        |   ph7 = p[p0x-d1, p0y, p0z-0.05, 0, 0, 0]
        | 
        |   # add the vertical touch points
        |   if pointtop[2] == 0:
        |     ph2up = p[ph2[0], ph2[1], ph2[2]+d3, ph2[3], ph2[4], ph2[5]]
        |     ph4up = p[ph4[0], ph4[1], ph4[2]+d3, ph4[3], ph4[4], ph4[5]]
        |   elif pointtop[2] > p0z + 0.914: # 0.914m = 36 inches
        |     ph2up = p[ph2[0], ph2[1], p0z + 0.914, ph2[3], ph2[4], ph2[5]]
        |     ph4up = p[ph4[0], ph4[1], p0z + 0.914, ph4[3], ph4[4], ph4[5]]
        |   else:
        |     ph2up = p[ph2[0], ph2[1], pointtop[2], ph2[3], ph2[4], ph2[5]]
        |     ph4up = p[ph4[0], ph4[1], pointtop[2], ph4[3], ph4[4], ph4[5]]
        |   end
        |   ret = struct(ph1=ph1, ph2=ph2, ph3=ph3, ph4=ph4, ph5=ph5, ph6=ph6, ph7=ph7, ph2up=ph2up, ph4up=ph4up)
        |   is_robot_at_reachable_spot(point0, ret)
        |   return ret
        | end
        | 
        | # this function checks whether the touchpoints are reachable AKA is the robot positioned in the right spot
        | # if everything looks good, it continues.
        | # if it detects a problem, it infinite loops a popup
        | def is_robot_at_reachable_spot(point0, struct_touchpoints):
        |   # first, check whether the corner is too low to the ground that the bottom homing will hit the ground (z < -400)
        |   lc_height = get_lift_column_height_condensed()
        |   # total height = zeroed lift column height (41.25 inches) (1.04775 m) plus lift column height plus robot relative height
        |   totalheight = 1.04775 + lc_height + point0[2]
        |   if totalheight < 1.04775 - 0.400:
        |     # bad
        |     popuptext = "Tank Corner is too low to the ground. Collisions will occur. Stop Program and raise tank. "
        |     # infinite loop
        |     while 1==1:
        |       popup(popuptext, title="Robot Positioning Warning",blocking=True)
        |     end
        |   end
        | 
        | 
        | 
        |   # next, check whether the touchpoints are reachable
        |   allvalid = check_structofpoints_validity(struct_touchpoints)
        |   if not allvalid:
        | 
        |     # then unreachable
        |     # generate message
        |     listproblems = ""
        |     listnames = ["ph1", "ph2", "ph3", "ph4", "ph5", "ph6", "ph7", "ph2up", "ph4up"]
        |     i = 0
        |     structlength = 9
        |     while i < structlength:
        |       curr = struct_touchpoints[i]
        |       valid = get_inverse_kin_has_solution(curr)
        |       if not valid:
        |         listproblems = listproblems + listnames[i]
        |       end
        |       i = i + 1
        |     end
        |     # display
        |     popuptext = "Robot is too far from tank corner. Cannot reach some necessary positions. Stop Program and move robot closer. " + listproblems
        |     # infinite loop
        |     while 1==1:
        |       popup(popuptext, title="Robot Positioning Warning",blocking=True)
        |     end
        |   end
        | 
        | end
        | 
        | # this function takes a struct of points as an argument, and checks whether every point in the list is reachable using get_inverse_kin_has_solution()
        | # this function does NOT check for weird twists or joint limits
        | # inputstruct must contain only points
        | # it returns true if all points are valid. it returns false if any points are valid
        | # a list of length 0 indicates that all points are valid
        | def check_structofpoints_validity(inputstruct):
        |   # next, check whether the touchpoints are reachable
        |   structlength = length(inputstruct)
        |   i = 0
        |   allvalid = True
        |   while i < structlength:
        |     curr = inputstruct[i]
        |     valid = get_inverse_kin_has_solution(curr)
        |     if not valid:
        |       return False
        |     end
        |     i = i + 1
        |   end
        |   return True
        | end
        | 
        | # checks the validity of all points during a left weld
        | # takes 2 arguments: struct1 (struct1[0] has to contain pointintersect) and struct2 (contains all the points (9) of the weld path)
        | def check_validity_left(struct1, struct2):
        |   #first, check whether robot is too close
        |   pointintersect = struct1[0]
        |   # next, check if the corner is too close to the robot to do a left around weld (complex but approximately X > -1300)
        |   # if y < 0, then x < -1300. if y < 480, then y > (1300+x)*8. if y > 480, then y > (1235+x)*4 + 500
        |   toocloseleftweld = False
        |   if pointintersect[1] < 0:
        |     if pointintersect[0] > -1.300:
        |       toocloseleftweld = True
        |     end
        |   elif pointintersect[1] < 0.480:
        |     if pointintersect[1] < (1.300 + pointintersect[0])*8:
        |       toocloseleftweld = True
        |     end
        |   else:
        |     if pointintersect[1] < (1.235 + pointintersect[0])*4 + 0.500:
        |       toocloseleftweld = True
        |     end
        |   end
        |   if toocloseleftweld:
        |     # bad
        |     popuptext = "Robot is too close to tank corner. Collisions may occur. Stop Program and move robot farther. "
        |     # infinite loop
        |     while 1==1:
        |       popup(popuptext, title="Robot Positioning Warning",blocking=True)
        |     end
        |   end
        | 
        |   #next, check whether all the points in the weldpath are valid
        |   structlength = 9
        |   i = 0
        |   allvalid = True
        |   listproblems = ""
        |   listnames = ["point1", "point2", "point4", "point5", "point_1", "point_2", "point_3", "point_4", "point_5"]
        |   while i < structlength:
        |     curr = struct2[i]
        |     valid = get_inverse_kin_has_solution(curr)
        |     if not valid:
        |       allvalid = False
        |       listproblems = listproblems + listnames[i]
        |     end
        |     i = i + 1
        |   end
        | 
        |   if not allvalid:
        |     # display
        |     popuptext = "Robot is too far from tank corner. Cannot reach some necessary positions. Stop Program and move robot closer. " + listproblems
        |     # infinite loop
        |     while 1==1:
        |       popup(popuptext, title="Robot Positioning Warning",blocking=True)
        |     end
        |   end
        | 
        |   # check whether the path involves weird turns or joint limits. currently just checks the first position
        |   p_prev = [-0.021118, -1.26292, 2.43578, 5.07088, -2.29912, 1.53362] #last point of left weld prerotate
        |   joints_1 = get_inverse_kin(struct2[0], p_prev) # struct2[0] is point1
        |   allGood = True
        |   i = 0
        |   structlength = 6
        |   while i < structlength:
        |     joint_curr = joints_1[i]
        |     # check for anything that exceeds joint limits
        |     degreesmax = 360 * pi / 180
        |     if joint_curr > degreesmax or joint_curr < degreesmax * -1:
        |       allGood = False
        |     end
        |     # check for anything that is significantly different than the aligned approach. could indicate a twist is needed. we dont want that
        |     maxdifference = 150 * pi / 180
        |     difference = joint_curr - p_prev[i]
        |     if difference > maxdifference or difference * -1 > maxdifference:
        |       allGood = False
        |     end
        |     i = i + 1
        |   end
        | 
        |   if not allGood:
        |     # call lift column extend function
        |     struct2 = floor_corner_lift_column_extend_left(struct2)
        | 
        |   end
        | 
        |   # return struct2 back
        |   return struct2
        | end
        | 
        | # checks the validity of all points during a right weld
        | def check_validity_right(struct1, struct2):
        |   # first, check whether the right pivot will bonk itself
        |   pointintersect = struct1[0]
        |   heading1 = struct1[1] # this is the direction that the welder will face when doing the right side of the box
        | 
        |   #first, check whether the heading is just too far offset
        |   # more than 15 degrees off of 45 is too much
        |   # normal heading is 216 degrees
        |   #201 degrees to 231 degrees
        |   heading1degrees = heading1 * 180 / pi
        |   if heading1degrees < 201 or heading1degrees > 231 :
        |     # then out of range
        |     popuptext = "Robot is not aligned at a 45 degree angle of corner (15 degree leeway). Collisions may occur. Stop Program and align robot. heading1degrees=" + str_cat("",heading1degrees)
        |     # infinite loop
        |     while 1==1:
        |       popup(popuptext, title="Robot Positioning Warning",blocking=True)
        |     end
        |   end
        | 
        |   #TODO: add the checks for whether x is too close, given the heading
        |   # add checks for whether x is too close, given the heading
        |   # different equations for whether heading offset > 5 degrees or less (inc. negative)
        |   headingoffset = heading1degrees - 216
        |   if headingoffset < 5:
        |     # then calculate a and b
        |     a = 0.4584 + -0.02369 * headingoffset
        |     b = (-1151.4 + 13.83 * headingoffset) / 1000
        |     # check whether x > a*y+b
        |     if pointintersect[0] > a * pointintersect[1] + b:
        |       # bad
        |       popuptext = "Robot is too close to tank corner or not at the right angle. Collisions may occur. Stop Program and align robot. "
        |       # infinite loop
        |       while 1==1:
        |         popup(popuptext, title="Robot Positioning Warning",blocking=True)
        |       end
        |     end
        |   else:
        |     # headingoffset > 5 degrees
        |     if pointintersect[1] < 0:
        |       if pointintersect[0] > -1150.0 / 1000.0:
        |         #bad
        |         popuptext = "Robot is too close to tank corner. Collisions may occur. Stop Program and align robot. "
        |         # infinite loop
        |         while 1==1:
        |           popup(popuptext, title="Robot Positioning Warning",blocking=True)
        |         end
        |       end
        |     else:
        |       # if x > .7736 y - 1101.9 then bad
        |       if pointintersect[0] > 0.7736 * pointintersect[1] - 1101.9 / 1000:
        |         popuptext = "Robot is too close to tank corner. Collisions may occur. Stop Program and align robot. "
        |         # infinite loop
        |         while 1==1:
        |           popup(popuptext, title="Robot Positioning Warning",blocking=True)
        |         end
        |       end
        |     end
        |   end
        | 
        |   #next, check whether all the points in the weldpath are valid
        |   structlength = 9
        |   i = 0
        |   allvalid = True
        |   listproblems = ""
        |   listnames = ["point1", "point2", "point4", "point5", "point_1", "point_2", "point_3", "point_4", "point_5"]
        |   while i < structlength:
        |     curr = struct2[i]
        |     valid = get_inverse_kin_has_solution(curr)
        |     if not valid:
        |       allvalid = False
        |       listproblems = listproblems + listnames[i]
        |     end
        |     i = i + 1
        |   end
        | 
        |   if not allvalid:
        |     # display
        |     popuptext = "Robot is too far from tank corner. Cannot reach some necessary positions. Stop Program and move robot closer. " + listproblems
        |     # infinite loop
        |     while 1==1:
        |       popup(popuptext, title="Robot Positioning Warning",blocking=True)
        |     end
        |   end
        | 
        |   # check whether the path involves weird turns or joint limits. currently just checks the first position
        |   p_prev = [-1.13307, -1.48911, 2.84785, 4.92357, -4.89059, 1.57184] #last point of right weld prerotate
        |   joints_1 = get_inverse_kin(struct2[0], p_prev) # struct2[0] is point1
        |   allGood = True
        |   i = 0
        |   structlength = 6
        |   while i < structlength:
        |     joint_curr = joints_1[i]
        |     # check for anything that exceeds joint limits
        |     degreesmax = 360 * pi / 180
        |     if joint_curr > degreesmax or joint_curr < degreesmax * -1:
        |       allGood = False
        |     end
        |     # check for anything that is significantly different than the aligned approach. could indicate a twist is needed. we dont want that
        |     maxdifference = 150 * pi / 180
        |     difference = joint_curr - p_prev[i]
        |     if difference > maxdifference or difference * -1 > maxdifference:
        |       allGood = False
        |     end
        |     i = i + 1
        |   end
        | 
        |   if not allGood:
        |     struct2 = floor_corner_lift_column_extend_right(struct2)
        |   end
        | 
        |   # return struct2 back
        |   return struct2
        | end
        | 
        | def floor_corner_lift_column_extend_right(struct2):
        |   # we know that p1 cannot be accessed without a twist
        |   # calculate the height needed to get to p1
        |   liftcolumnincrement = 2.0 # mm
        |   enoughHeightAdded = False
        |   liftColumnHeightTest = 0
        |   while not enoughHeightAdded:
        |     liftColumnHeightTest = liftColumnHeightTest + liftcolumnincrement
        |     # set the orig_joints for p1. p1 demo was joint angles of [-0.45, -31.79, 56.47, 333.06, -130.98, 87.87] (degrees)
        |     # which equals [-0.007853981633974475, -0.5548401692089968, 0.985587428601197, 5.812993606692308, -2.28603225426217, 1.5336208137274159]
        |     orig_joints = [-0.007853981633974475, -0.5548401692089968, 0.985587428601197, 5.812993606692308, -2.28603225426217, 1.5336208137274159]
        |     # get the modified point:
        |     origp1 = struct2[0]
        |     testp1 = p[origp1[0], origp1[1], origp1[2] - liftColumnHeightTest / 1000.0, origp1[3], origp1[4], origp1[5]]
        |     testpa1 = p[origp1[0]+0.05, origp1[1]+0.05, origp1[2] - liftColumnHeightTest / 1000, origp1[3], origp1[4], origp1[5]]
        |     enoughHeightAdded = can_pose_be_reached_without_twist(testp1, orig_joints) and can_pose_be_reached_without_twist(testpa1, orig_joints)
        |   end
        | 
        |   origp2 = struct2[1]
        |   testp2 = p[origp2[0], origp2[1], origp2[2] - liftColumnHeightTest / 1000.0, origp2[3], origp2[4], origp2[5]]
        |   origp4 = struct2[2]
        |   testp4 = p[origp4[0], origp4[1], origp4[2] - liftColumnHeightTest / 1000, origp4[3], origp4[4], origp4[5]]
        |   origp5 = struct2[3]
        |   testp5 = p[origp5[0], origp5[1], origp5[2] - liftColumnHeightTest / 1000, origp5[3], origp5[4], origp5[5]]
        | 
        | 
        | 
        |   liftcolumnzneeded = liftColumnHeightTest
        |   ret = struct(point1=testp1,point2=testp2,point4=testp4,point5=testp5,point_1=struct2[4],point_2=struct2[5],point_3=struct2[6],point_4=struct2[7],point_5=struct2[8])
        |   return ret
        | 
        | end
        | 
        | # this function gets called if you are doing a left floor corner extended, and the top is too high to reach (twists, etc.)
        | # this function takes the struct2 of weld points and modifies them (by subtracting from z) until the first weld point is reachable.
        | # it determines the height that the lift column needs to raise to make the first point reachable
        | # it then checks whether that height will allow the other points to be reachable
        | # if its all good, it sets the global variable liftcolumnzneeded, modifies struct2's points, and returns struct2
        | # if its not all good, then it displays an error message popup.
        | def floor_corner_lift_column_extend_left(struct2):
        |   # we know that p1 cannot be accessed without a twist
        |   # calculate the height needed to get to p1
        |   liftcolumnincrement = 2 # mm
        |   enoughHeightAdded = False
        |   liftColumnHeightTest = 0
        |   while not enoughHeightAdded:
        |     liftColumnHeightTest = liftColumnHeightTest + liftcolumnincrement
        |     # set the orig_joints for p1. p1 demo was joint angles of [-0.45, -31.79, 56.47, 333.06, -130.98, 87.87] (degrees)
        |     # which equals [-0.007853981633974475, -0.5548401692089968, 0.985587428601197, 5.812993606692308, -2.28603225426217, 1.5336208137274159]
        |     orig_joints = [-0.007853981633974475, -0.5548401692089968, 0.985587428601197, 5.812993606692308, -2.28603225426217, 1.5336208137274159]
        |     # get the modified point:
        |     origp1 = struct2[0]
        |     testp1 = p[origp1[0], origp1[1], origp1[2] - liftColumnHeightTest / 1000, origp1[3], origp1[4], origp1[5]]
        |     enoughHeightAdded = can_pose_be_reached_without_twist(testp1, orig_joints)
        |   end
        | 
        |   # check whether the other 3 points are valid
        |   valid = True
        |   # get the modified point
        |   origp2 = struct2[1]
        |   testp2 = p[origp2[0], origp2[1], origp2[2] - liftColumnHeightTest / 1000, origp2[3], origp2[4], origp2[5]]
        |   # p2 demo was joint angles of [-0.45, -21.2, 56.98, 321.95, -130.97, 87.85] (degrees)
        |   # which equals [-0.007853981633974475, -0.3700098014227975, 0.9944886077863679, 5.619087526795738, -2.285857721336971, 1.5332717478770168]
        |   orig_joints = [-0.007853981633974475, -0.3700098014227975, 0.9944886077863679, 5.619087526795738, -2.285857721336971, 1.5332717478770168]
        |   valid = valid and can_pose_be_reached_without_twist(testp2, orig_joints)
        |   # get the modified point
        |   origp4 = struct2[2]
        |   testp4 = p[origp4[0], origp4[1], origp4[2] - liftColumnHeightTest / 1000, origp4[3], origp4[4], origp4[5]]
        |   # p4 demo was joint angles of [-8.62, -43.23, 99.53, 213.86, -89.19, 40.78] (degrees)
        |   # which equals [-0.15044738152191103, -0.7545058356371478, 1.7371262045099545, 3.7325611383150696, -1.556659159853741, 0.7117452689632868]
        |   orig_joints = [-0.15044738152191103, -0.7545058356371478, 1.7371262045099545, 3.7325611383150696, -1.556659159853741, 0.7117452689632868]
        |   valid = valid and can_pose_be_reached_without_twist(testp4, orig_joints)
        |   # get the modified point
        |   origp5 = struct2[3]
        |   testp5 = p[origp5[0], origp5[1], origp5[2] - liftColumnHeightTest / 1000, origp5[3], origp5[4], origp5[5]]
        |   # p5 demo was joint angles of [-0.59, -34.36, 77.71, 226.7, -89.18, 48.81] (degrees)
        |   # which equals [-0.010297442586766533, -0.5996951309852511, 1.356295361724792, 3.9566614142711405, -1.5564846269285415, 0.8518952078984314]
        |   orig_joints = [-0.010297442586766533, -0.5996951309852511, 1.356295361724792, 3.9566614142711405, -1.5564846269285415, 0.8518952078984314]
        |   valid = valid and can_pose_be_reached_without_twist(testp5, orig_joints)
        | 
        |   if not valid:
        |     # display
        |     popuptext = "Top of Weld is too high above robot. Cannot reach some necessary positions. Stop Program and try again with a lower top point. "
        |     # infinite loop
        |     while 1==1:
        |       popup(popuptext, title="Robot Positioning Warning",blocking=True)
        |     end
        |   else:
        |     liftcolumnzneeded = liftColumnHeightTest
        |     ret = struct(point1=testp1,point2=testp2,point4=testp4,point5=testp5,point_1=struct2[4],point_2=struct2[5],point_3=struct2[6],point_4=struct2[7],point_5=struct2[8])
        |     return ret
        |   end
        | end
        | 
        | # this function calculates whether a given pose can be reached, and if it can, whether it requires a wrist twist (from the seed joint angles)
        | # arguments are target pose (p[x,y,z,rx,ry,rz]) and orig_joints which is the 6 joint angles of a pose that is close by the target pose and has the desired joint angles
        | # returns true if the pose is valid and requires no twist. If pose is valid but requires a twist, returns false. If pose is invalid, returns false.
        | def can_pose_be_reached_without_twist(pose, orig_joints):
        |   # first, determine if the pose is valid
        |   valid = get_inverse_kin_has_solution(pose)
        |   if not valid:
        |     return False
        |   end
        |   joints_1 = get_inverse_kin(pose, orig_joints)
        |   #iterate through the 6 joints
        |   allGood = True
        |   i = 0
        |   structlength = 6
        |   while i < structlength:
        |     joint_curr = joints_1[i]
        |     # check for anything that exceeds joint limits
        |     degreesmax = 360 * pi / 180
        |     if joint_curr > degreesmax or joint_curr < degreesmax * -1:
        |       allGood = False
        |     end
        |     # check for anything that is significantly different than the aligned approach. could indicate a twist is needed. we dont want that
        |     maxdifference = 150 * pi / 180
        |     difference = joint_curr - orig_joints[i]
        |     if difference > maxdifference or difference * -1 > maxdifference:
        |       allGood = False
        |     end
        |     i = i + 1
        |   end
        |   return allGood
        | end
        | 
        | # this function sends a signal to turn extrusion on
        | def turn_extrusion_on():
        |   # flush the channel
        |   resp0 = send_serial_signal(["u", "r", "?"])
        |   # send the signal
        |   resp1 = send_serial_signal(["u", "R", "1"])
        |   # if resp <> "uR1"
        |   if resp1 != [252,82,49]:
        |     # turn off extrusion and heating. inform calvin
        |     resp2 = send_serial_signal(["u", "R", "0"])
        |     resp3 = send_serial_signal(["u", "H", "0"])
        |     popuptext = "Error code encountered while trying to start extrusion. Find Calvin. "
        |     while 1==1:
        |       popup(popuptext, title="Extrusion Error Code",blocking=True)
        |       popup(resp1, blocking=True)
        |     end
        |   end
        | end
        | 
        | # this function sends a signal and receives a response
        | # signal is a list of 3 strings, 1 character each. first is u. second is the next character. third is final character
        | def send_serial_signal(signal):
        |   signal2char = signal[1]
        |   signal3char = signal[2]
        |   listsignal = [252, get_corr_number(signal2char), get_corr_number(signal3char)]
        |   resp1 = WTSerialBridge.send_command("/dev/ttyUSB0",1200, 8, "None", "One", "None", 1000, "None", "None", listsignal, True)
        |   return resp1
        | end
        | 
        | # this function converts a letter into its ascii number
        | def get_corr_number(letter):
        |   if letter == "A":
        |     return 65
        |   elif letter == "H":
        |     return 72
        |   elif letter == "R":
        |     return 82
        |   elif letter == "M":
        |     return 77
        |   elif letter == "E":
        |     return 69
        |   elif letter == "a":
        |     return 97
        |   elif letter == "b":
        |     return 98
        |   elif letter == "h":
        |     return 104
        |   elif letter == "r":
        |     return 114
        |   elif letter == "s":
        |     return 115
        |   elif letter == "m":
        |     return 109
        |   elif letter == "0":
        |     return 48
        |   elif letter == "1":
        |     return 49
        |   elif letter == "2":
        |     return 50
        |   elif letter == "3":
        |     return 51
        |   elif letter == "4":
        |     return 52
        |   elif letter == "5":
        |     return 53
        |   elif letter == "6":
        |     return 54
        |   elif letter == "7":
        |     return 55
        |   elif letter == "8":
        |     return 56
        |   elif letter == "9":
        |     return 57
        |   elif letter == "?":
        |     return 63
        |   end
        | end
        | 
        | # this function checks whether the welder is in the ready state.
        | # to be called at the beginning of Main Program
        | def welder_state_ready():
        |   # flush the channel
        |   resp0 = send_serial_signal(["u", "s", "?"])
        |   # send the signal
        |   resp1 = send_serial_signal(["u", "s", "?"])
        |   # if resp1 == [252,115,49] (us1) then it is ready. otherwise, it is not
        |   if resp1 != [252,115,49]:
        |     popuptext = "Welder is not ready for extrusion. Follow the instructions to start heating welder. "
        |     while 1==1:
        |       popup(popuptext, title="Welder Not Ready",blocking=True)
        |     end
        |   end
        | 
        | end
        | 
        | def get_lift_column_height():
        |   # begin: URCap Program Node
        |   #   Source: MachineLogic for Universal Robots, 3.1.7, Vention Inc.
        |   #   Type: MachineLogic for Universal Robots
        |   #$ 5 "MachineLogic Get Position"
        |   while isVentionMovementBusyMachineMotion1==True:
        |     sleep(0.05)
        |   end
        |   if(isVentionMovementBusyMachineMotion1 == False):
        |     isVentionMovementBusyMachineMotion1 = True
        |     socket_send_string("estop/status;", "MachineMotion1")
        |     temp_estop_var_vention = socket_read_string("MachineMotion1",timeout=15)
        |     while(temp_estop_var_vention=="estop/status true"):
        |       if temp_estop_var_vention=="estop/status true":
        |         sendStringWithTimeout("estop/systemreset/request","Ack estop/systemreset/request;","MachineMotion1")
        |       end
        |       socket_send_string("estop/status;", "MachineMotion1")
        |       temp_estop_var_vention = socket_read_string("MachineMotion1",timeout=15)
        |       if temp_estop_var_vention=="estop/status true":
        |         popup("MachineMotion in estop, make sure you have all emergency modules released manually. If you continue the system will try to reset MachineMotion automatically.",blocking=True)
        |       end
        |     end
        |   else:
        |     popup("resource is being used already: MachineMotion1")
        |     halt
        |   end
        |   socket_send_string("GET im_get_controller_pos_axis_1;", "MachineMotion1")
        |   temp_drive = socket_read_ascii_float(1, "MachineMotion1",timeout=15)
        |   global var_1 = temp_drive[1]
        |   isVentionMovementBusyMachineMotion1 = False
        |   sleep(0.03)
        |   # end: URCap Program Node
        | end
        | 
        | def get_lift_column_height_condensed():
        |   socket_send_string("GET im_get_controller_pos_axis_1;", "MachineMotion1")
        |   temp_drive = socket_read_ascii_float(1, "MachineMotion1",timeout=15)
        |   ret = temp_drive[1]
        |   return ret
        | end
  'list possible points'
  Folder robot 1 moves
    If 1≟2
      MoveJ speed 60 deg/s, acceleration 80 deg/s^2 (useActiveTCP=true optimoveEnabled=false optiMoveSpeed=0.3 optiMoveAcceleration=0.09) feature=Base
        Waypoint r1_ek_oldhome: TCP in base x=397.38 y=356.254 z=319.821 mm, rx=2.3163 ry=2.0576 rz=0.0741 rad; joints [-198.126, -117.851, 133.303, -13.009, -11.422, -6.035] deg; TCP offset x=-5.49 y=-328 z=106.39 mm, rx=1.2092 ry=-1.2092 rz=1.2092 rad
        Waypoint r1_ek_extrude: TCP in base x=454.852 y=405.449 z=64.015 mm, rx=2.3168 ry=2.0514 rz=0.0767 rad; joints [-187.624, -89.406, 141.395, -19.732, -0.818, -36.116] deg
        Waypoint r1_ek_front: TCP in base x=439.065 y=405.452 z=65.996 mm, rx=2.3168 ry=2.0514 rz=0.0766 rad; joints [-187.962, -93.321, 143.386, -27.168, -1.131, -26.752] deg
        Waypoint r1_ek_middle: TCP in base x=419.01 y=404.851 z=65.995 mm, rx=2.3096 ry=2.0447 rz=0.0891 rad; joints [-188.553, -97.485, 146.002, -33.769, -1.69, -19.324] deg
        Waypoint r1_ek_middle2: TCP in base x=417.012 y=405.435 z=65.003 mm, rx=2.3169 ry=2.0513 rz=0.0766 rad; joints [-188.493, -97.025, 145.794, -33.21, -1.638, -19.415] deg
        Waypoint r1_ek_bottom: TCP in base x=413.072 y=405.431 z=68 mm, rx=2.3168 ry=2.0513 rz=0.0767 rad; joints [-188.596, -97.887, 146.02, -33.517, -1.738, -18.475] deg
        Waypoint r1_ek_end: TCP in base x=389.999 y=405.444 z=68.005 mm, rx=2.3169 ry=2.0514 rz=0.0766 rad; joints [-189.248, -101.07, 148.002, -36.337, -2.38, -14.447] deg
  Folder robot 2 moves
    If 1≟2
      MoveJ speed 60 deg/s, acceleration 80 deg/s^2 (useActiveTCP=true optimoveEnabled=false optiMoveSpeed=0.3 optiMoveAcceleration=0.09) feature=Base
        Waypoint r2_ek_oldhome: TCP in base x=397.38 y=356.254 z=319.821 mm, rx=2.3163 ry=2.0576 rz=0.0741 rad; joints [-198.308, -118.162, 133.451, -12.562, -11.515, -6.325] deg; TCP offset x=-9.5 y=-328 z=105.73 mm, rx=1.2092 ry=-1.2092 rz=1.2092 rad
        SuppressedNode
          Waypoint Waypoint_1: TCP in base x=612.886 y=429.305 z=100.477 mm, rx=1.8619 ry=2.4807 rz=0.0957 rad; joints [-182.793, -81.736, 125.569, -42.478, -18.966, -5.44] deg
        Waypoint r2_ek_extrude: TCP in base x=612.886 y=429.305 z=100.477 mm, rx=2.15 ry=2.2258 rz=0.0874 rad; joints [-183.316, -85.158, 129.692, -39.696, -5.262, -8.969] deg
        Waypoint r2_ek_front: TCP in base x=556.405 y=429.305 z=76.984 mm, rx=-2.1704 ry=-2.2682 rz=-0.0159 rad; joints [-183.513, -85.623, 132.794, -41.666, -5.994, -5.809] deg
        Waypoint r2_ek_middle: TCP in base x=550.034 y=429.305 z=76.254 mm, rx=-2.1704 ry=-2.2682 rz=-0.0159 rad; joints [-183.554, -85.983, 133.283, -41.831, -6.035, -5.773] deg
        Waypoint r2_ek_bottom: TCP in base x=546.595 y=429.305 z=80.868 mm, rx=-2.1704 ry=-2.2682 rz=-0.0159 rad; joints [-183.576, -86.513, 133.34, -41.373, -6.058, -5.758] deg
        Waypoint r2_ek_end: TCP in base x=537.335 y=429.305 z=80.868 mm, rx=-2.1704 ry=-2.2682 rz=-0.0159 rad; joints [-183.639, -87.118, 134.001, -41.482, -6.12, -5.705] deg
  'detemine correct points for which robot'
  If robot_number≟1
    Folder robot1 positions
      ek_oldhome := r1_ek_oldhome_p
      ek_extrude := r1_ek_extrude_p
      ek_front := r1_ek_front_p
      ek_middle := r1_ek_middle_p
      ek_middle2 := r1_ek_middle2_p
      ek_bottom := r1_ek_bottom_p
      ek_end := r1_ek_end_q
  ElseIf robot_number≟2
    Folder robot1 positions
      ek_oldhome := r2_ek_oldhome_p
      ek_extrude := r2_ek_extrude_p
      ek_front := r2_ek_front_p
      ek_middle := r2_ek_middle_p
      ek_middle2 := r2_ek_middle_p
      ek_bottom := r2_ek_bottom_p
      ek_end := r2_ek_end_q
  'start of program'
  SuppressedNode
    SafeHome (positionOptionType=SPEED_AND_ACCELERATION speed=1.047198 acceleration=1.396263 nextMotionTime=2)
  Set NoAction tcp=pretend_welder
  MoveJ speed 60 deg/s, acceleration 80 deg/s^2 (useActiveTCP=true optimoveEnabled=false optiMoveSpeed=0.3 optiMoveAcceleration=0.09) feature=Base
    SuppressedNode
      Waypoint r1_ek_oldhome: TCP in base x=397.38 y=356.254 z=319.821 mm, rx=2.3163 ry=2.0576 rz=0.0741 rad; joints [-198.126, -117.851, 133.303, -13.009, -11.422, -6.035] deg; TCP offset x=-5.49 y=-328 z=106.39 mm, rx=1.2092 ry=-1.2092 rz=1.2092 rad
    Waypoint Variable (Variable): variable=ek_oldhome
    'above waypoint is home'
  'move above bucket'
  MoveJ speed 60 deg/s, acceleration 80 deg/s^2 (useActiveTCP=true optimoveEnabled=false optiMoveSpeed=0.3 optiMoveAcceleration=0.09) feature=Base
    SuppressedNode
      Waypoint r1_ek_extrude: TCP in base x=454.852 y=405.449 z=64.015 mm, rx=2.3168 ry=2.0514 rz=0.0767 rad; joints [-187.624, -89.406, 141.395, -19.732, -0.818, -36.116] deg
    Waypoint Variable (Variable): variable=ek_extrude
  'extrude out a foot'
  SuppressedNode
    Script: turn_extrusion_on()
  URCap WireTank Serial (WireTank Serial, WireTank, LLC) dataModel(NODE_TITLE=Serial Bridge uR1, Command=[252,82,49], QUERY=false, byte_array=true, OUTPUT_ENTRY=Static, Variable(key=OUTPUT_VARIABLE, variable(name=HwResp)))
  Set DigitalOutput pin=digital_out[0]; digitalValue=1
  Wait Sleep waitTime=24
  URCap WireTank Serial (WireTank Serial, WireTank, LLC) dataModel(QUERY=false, NODE_TITLE=Serial Bridge uR0, Command=[252,82,48], byte_array=true, OUTPUT_ENTRY=Static, Variable(key=OUTPUT_VARIABLE, variable(name=HwResp)))
  Wait Sleep waitTime=1
  Set DigitalOutput pin=digital_out[0]; digitalValue=0
  'slice'
  MoveL speed 30 mm/s, acceleration 50 mm/s^2 (useActiveTCP=true optimoveEnabled=false optiMoveSpeed=0.3 optiMoveAcceleration=0.09) feature=Base
    SuppressedNode
      Waypoint r1_ek_front: TCP in base x=439.065 y=405.452 z=65.996 mm, rx=2.3168 ry=2.0514 rz=0.0766 rad; joints [-187.962, -93.321, 143.386, -27.168, -1.131, -26.752] deg
    SuppressedNode
      Waypoint r1_ek_middle: TCP in base x=419.01 y=404.851 z=65.995 mm, rx=2.3096 ry=2.0447 rz=0.0891 rad; joints [-188.553, -97.485, 146.002, -33.769, -1.69, -19.324] deg
    SuppressedNode
      Waypoint r1_ek_middle2: TCP in base x=417.012 y=405.435 z=65.003 mm, rx=2.3169 ry=2.0513 rz=0.0766 rad; joints [-188.493, -97.025, 145.794, -33.21, -1.638, -19.415] deg
    SuppressedNode
      Waypoint r1_ek_bottom: TCP in base x=413.072 y=405.431 z=68 mm, rx=2.3168 ry=2.0513 rz=0.0767 rad; joints [-188.596, -97.887, 146.02, -33.517, -1.738, -18.475] deg
    SuppressedNode
      Waypoint r1_ek_end: TCP in base x=389.999 y=405.444 z=68.005 mm, rx=2.3169 ry=2.0514 rz=0.0766 rad; joints [-189.248, -101.07, 148.002, -36.337, -2.38, -14.447] deg
    Waypoint Variable (Variable): variable=ek_front
    Waypoint Variable (Variable): variable=ek_middle
    Waypoint Variable (Variable): variable=ek_middle2
    Waypoint Variable (Variable): variable=ek_bottom
    Waypoint Variable (Variable): variable=ek_end
  MoveJ speed 60 deg/s, acceleration 80 deg/s^2 (useActiveTCP=true optimoveEnabled=false optiMoveSpeed=0.3 optiMoveAcceleration=0.09) feature=Base
    SuppressedNode
      Waypoint r1_ek_oldhome: TCP in base x=397.38 y=356.254 z=319.821 mm, rx=2.3163 ry=2.0576 rz=0.0741 rad; joints [-198.126, -117.851, 133.303, -13.009, -11.422, -6.035] deg
    Waypoint Variable (Variable): variable=ek_oldhome
    'above waypoint is home'
  SuppressedNode
    SafeHome (positionOptionType=SPEED_AND_ACCELERATION speed=1.047198 acceleration=1.396263 nextMotionTime=2)
SubProgram align_tcp_forward (keepSynchronizedWithDisk=false) programFile=/programs/align_tcp_forward.urp
  'this program aligns the tcp parallel to the y direction'
  cp := get_actual_tcp_pose()
  aligned_y_pose := p[cp[0],cp[1],cp[2],0,-1.570796,0]
  MoveJ speed 60 deg/s, acceleration 80 deg/s^2 (useActiveTCP=true optimoveEnabled=false optiMoveSpeed=0.3 optiMoveAcceleration=0.09) feature=Base
    Waypoint Variable (Variable): variable=aligned_y_pose
SubProgram align_tcp_up (keepSynchronizedWithDisk=false) programFile=/programs/align_tcp_up.urp
  'this program aligns the tcp parallel to the y direction'
  cp := get_actual_tcp_pose()
  aligned_y_pose := p[cp[0],cp[1],cp[2],0,0,0]
  MoveJ speed 60 deg/s, acceleration 80 deg/s^2 (useActiveTCP=true optimoveEnabled=false optiMoveSpeed=0.3 optiMoveAcceleration=0.09) feature=Base
    Waypoint Variable (Variable): variable=aligned_y_pose
SubProgram align_for_step (keepSynchronizedWithDisk=false) programFile=/programs/align_for_step.urp
  'first move block is unnecessay and bad'
  SuppressedNode
    MoveJ speed 60 deg/s, acceleration 80 deg/s^2 (useActiveTCP=true optimoveEnabled=false optiMoveSpeed=0.3 optiMoveAcceleration=0.09) feature=Base
      'belowis oldhome'
      Waypoint Waypoint_1: TCP in base x=397.354 y=356.263 z=319.809 mm, rx=2.3163 ry=2.0576 rz=0.0741 rad; joints [-198.308, -118.162, 133.452, -12.561, -11.517, -6.326] deg; TCP offset x=-9.5 y=-328 z=105.73 mm, rx=1.2092 ry=-1.2092 rz=1.2092 rad
      SuppressedNode
        Waypoint Waypoint_2: TCP in base x=102.072 y=804.129 z=-21.158 mm, rx=-1.0098 ry=-2.9661 rz=0.0347 rad; joints [-131.791, -72.228, 126.432, -52.794, -4.122, -0.058] deg
      SuppressedNode
        Waypoint Waypoint_3: TCP in base x=-481.576 y=738.776 z=-387.745 mm, rx=-0.0268 ry=3.1371 rz=-0.1325 rad; joints [-88.373, -42.244, 121.849, -79.055, 0.705, 4.289] deg
      Waypoint Waypoint_4: TCP in base x=-790.625 y=220.046 z=-730.503 mm, rx=-0.9425 ry=2.9648 rz=-0.1356 rad; joints [-49.775, -15.59, 117.776, -102.401, 4.996, 5.448] deg
      Waypoint Waypoint_5: TCP in base x=-802.158 y=237.168 z=-730.663 mm, rx=0.8868 ry=-2.4516 rz=0.2829 rad; joints [-61.24, 14.733, 101.407, -222.645, 33.575, 110.967] deg
      Waypoint Waypoint_6: TCP in base x=-687.678 y=589.975 z=-233.622 mm, rx=-0.3444 ry=-1.0001 rz=-2.0808 rad; joints [-61.24, 14.733, 101.407, -222.645, 33.575, -30.853] deg
      SuppressedNode
        Waypoint goalpt: TCP in base x=-796.965 y=229.005 z=-75.004 mm, rx=0 ry=0 rz=-2.526 rad; joints [-49.775, -15.59, 117.776, -102.401, 4.996, -179.788] deg
      Waypoint goalpt2: TCP in base x=-1080.054 y=352.633 z=-86.722 mm, rx=0.0341 ry=-0.0008 rz=-2.631 rad; joints [-41.761, 5.394, 77.547, 101.81, -19.08, -4.137] deg
      Waypoint dummythere: TCP in base x=-1288.589 y=229.005 z=-75.004 mm, rx=0 ry=0 rz=-2.526 rad; joints [-29.748, -12.575, 79.071, -66.58, 25.031, -179.927] deg
  'second one is good'
  SuppressedNode
    MoveJ speed 60 deg/s, acceleration 80 deg/s^2 (useActiveTCP=true optimoveEnabled=false optiMoveSpeed=0.3 optiMoveAcceleration=0.09) feature=Base
      Waypoint goalpt2: TCP in base x=-1080.054 y=352.633 z=-86.722 mm, rx=0.0341 ry=-0.0008 rz=-2.631 rad; joints [-41.761, 5.394, 77.547, 101.81, -19.08, -4.137] deg
  'above was for wrong weldpath'
  SuppressedNode
    Folder savepoints
      MoveJ speed 60 deg/s, acceleration 80 deg/s^2 (useActiveTCP=true optimoveEnabled=false optiMoveSpeed=0.3 optiMoveAcceleration=0.09) feature=Base
        Waypoint leftstart: TCP in base x=-1168.534 y=251.879 z=303.712 mm, rx=-1.4388 ry=-0.6695 rz=0.6003 rad; joints [-161.388, -128.913, -89.606, -145.038, 61.894, 92.57] deg
  SuppressedNode
    MoveJ speed 60 deg/s, acceleration 80 deg/s^2 (useActiveTCP=true optimoveEnabled=false optiMoveSpeed=0.3 optiMoveAcceleration=0.09) feature=Base
      'final point before pa1'
      Waypoint Waypoint_7: TCP in base x=-913.411 y=251.879 z=303.712 mm, rx=-1.2351 ry=-1.1043 rz=1.0523 rad; joints [-156.391, -105.358, -132.178, -128.187, 33.298, 95.672] deg
      'oldhome'
      Waypoint Waypoint_8: TCP in base x=397.354 y=356.263 z=319.809 mm, rx=2.3163 ry=2.0576 rz=0.0741 rad; joints [-198.308, -118.162, 133.452, -12.561, -11.517, -6.326] deg
  MoveJ speed 60 deg/s, acceleration 80 deg/s^2 (useActiveTCP=true optimoveEnabled=false optiMoveSpeed=0.3 optiMoveAcceleration=0.09) feature=Base
    'from oldhome, actual path'
    SuppressedNode
      Waypoint Waypoint_9: TCP in base x=683.137 y=304.628 z=775.294 mm, rx=1.9572 ry=1.7212 rz=0.4516 rad; joints [-193.46, -116.682, 102.732, -25.933, -6.334, 5.47] deg
    SuppressedNode
      Waypoint Waypoint_10: TCP in base x=-197.847 y=491.143 z=1723.576 mm, rx=-0.0125 ry=0.2444 rz=1.7982 rad; joints [-175.692, -50.406, -94.795, -74.947, 12.663, 48.707] deg
    Waypoint Waypoint_1: TCP in base x=-557.589 y=419.56 z=1207.727 mm, rx=-0.5026 ry=-0.0558 rz=1.8139 rad; joints [-165.719, -50.766, -121.227, -102.266, 18.039, 76.633] deg
    SuppressedNode
      Waypoint Waypoint_12: TCP in base x=-793.876 y=251.879 z=303.712 mm, rx=-1.2351 ry=-1.1043 rz=1.0523 rad; joints [-150.736, -98.884, -141.754, -124.357, 38.932, 94.772] deg
  MoveJ speed 60 deg/s, acceleration 80 deg/s^2 (useActiveTCP=true optimoveEnabled=false optiMoveSpeed=0.3 optiMoveAcceleration=0.09) feature=Base
    SuppressedNode
      Waypoint Waypoint_12: TCP in base x=-793.876 y=251.879 z=303.712 mm, rx=-1.2351 ry=-1.1043 rz=1.0523 rad; joints [-150.736, -98.884, -141.754, -124.357, 38.932, 94.772] deg
    Waypoint Waypoint_3: TCP in base x=-479.957 y=297.468 z=291.375 mm, rx=-0.7812 ry=-1.774 rz=1.7129 rad; joints [-222.662, -82.07, -155.488, -122.893, -85.563, 87.81] deg
  SuppressedNode
    Folder dummy points
      'for seeing if it goes to each side correctly'
      MoveJ speed 60 deg/s, acceleration 80 deg/s^2 (useActiveTCP=true optimoveEnabled=false optiMoveSpeed=0.3 optiMoveAcceleration=0.09) feature=Base
        'right side weld'
        Waypoint Waypoint_15: TCP in base x=-1072.479 y=376.012 z=295.965 mm, rx=-0.7812 ry=-1.774 rz=1.7129 rad; joints [-196.962, -109.785, -121.389, -129.338, -59.875, 88.022] deg
      MoveL speed 10 mm/s, acceleration 50 mm/s^2 (useActiveTCP=true optimoveEnabled=false optiMoveSpeed=0.3 optiMoveAcceleration=0.09) feature=Base
        Waypoint Waypoint_14: TCP in base x=-1156.816 y=297.468 z=291.375 mm, rx=-0.7812 ry=-1.774 rz=1.7129 rad; joints [-189.786, -111.954, -118.346, -130.254, -52.7, 88.101] deg
SubProgram retreat_from_step (keepSynchronizedWithDisk=false) programFile=/programs/retreat_from_step.urp
  SuppressedNode
    Folder dummy points
      MoveJ speed 60 deg/s, acceleration 80 deg/s^2 (useActiveTCP=true optimoveEnabled=false optiMoveSpeed=0.3 optiMoveAcceleration=0.09) feature=Base
        'right side end points'
        Waypoint Waypoint_1: TCP in base x=-1253.519 y=364.13 z=-67.585 mm, rx=0.018 ry=0.0176 rz=0.7803 rad; joints [-179.095, -181.39, -36.733, -141.231, 46.177, 180.871] deg
        Waypoint Waypoint_3: TCP in base x=-1253.519 y=364.13 z=-129.324 mm, rx=0.018 ry=0.0176 rz=0.7803 rad; joints [-179.093, -185.871, -31.706, -141.776, 46.177, 180.869] deg
      MoveJ speed 60 deg/s, acceleration 80 deg/s^2 (useActiveTCP=true optimoveEnabled=false optiMoveSpeed=0.3 optiMoveAcceleration=0.09) feature=Base
        'left side end points'
        Waypoint Waypoint_4: TCP in base x=-1258.059 y=209.945 z=-65.388 mm, rx=0.0265 ry=-0.0276 rz=2.2505 rad; joints [-170.66, -165.644, -86.102, -104.787, -29.65, 176.354] deg
        Waypoint Waypoint_5: TCP in base x=-1258.059 y=209.945 z=-131.718 mm, rx=0.0265 ry=-0.0276 rz=2.2505 rad; joints [-170.658, -169.867, -82.992, -103.675, -29.649, 176.354] deg
  MoveJ speed 60 deg/s, acceleration 80 deg/s^2 (useActiveTCP=true optimoveEnabled=false optiMoveSpeed=0.3 optiMoveAcceleration=0.09) feature=Base
    Waypoint Waypoint_16: TCP in base x=-670.966 y=326.422 z=-178.215 mm, rx=0.0098 ry=0.0257 rz=1.6447 rad; joints [-167.814, -172.971, -116.48, -67.413, 7.981, 178.204] deg
  MoveJ speed 60 deg/s, acceleration 80 deg/s^2 (useActiveTCP=true optimoveEnabled=false optiMoveSpeed=0.3 optiMoveAcceleration=0.09) feature=Base
    Waypoint Waypoint_17: TCP in base x=-635.85 y=491.712 z=259.684 mm, rx=-0.4995 ry=-0.7883 rz=1.854 rad; joints [-203.235, -128.315, -150.467, -80.055, -46.632, 133.613] deg
    Waypoint Waypoint_18: TCP in base x=-479.957 y=297.468 z=291.375 mm, rx=-0.7812 ry=-1.774 rz=1.7129 rad; joints [-222.662, -82.07, -155.488, -122.893, -85.563, 87.81] deg
  MoveJ speed 60 deg/s, acceleration 80 deg/s^2 (useActiveTCP=true optimoveEnabled=false optiMoveSpeed=0.3 optiMoveAcceleration=0.09) feature=Base
    Waypoint Waypoint_20: TCP in base x=-557.589 y=419.56 z=1207.727 mm, rx=-0.5026 ry=-0.0558 rz=1.8139 rad; joints [-165.719, -50.766, -121.227, -102.266, 18.039, 76.633] deg
  SafeHome (positionOptionType=SPEED_AND_ACCELERATION speed=1.047198 acceleration=1.396263 nextMotionTime=2)
SubProgram Corner_Homing_45 (keepSynchronizedWithDisk=false) programFile=/programs/Corner Homing 45.urp
  'Use this program when tool is already positioned close to corner at 45deg'
  'tool flange will seek all 3 sides. will save those 5 locs in p__'
  Set NoAction tcp=pretend_w_top
  'dummy move below for debug'
  SuppressedNode
    SafeHome (positionOptionType=SPEED_AND_ACCELERATION speed=1.047198 acceleration=1.396263 nextMotionTime=2)
  SuppressedNode
    MoveJ speed 60 deg/s, acceleration 80 deg/s^2 (useActiveTCP=true optimoveEnabled=false optiMoveSpeed=0.3 optiMoveAcceleration=0.09) feature=Base
      Waypoint Waypoint_1: TCP in base x=-726.76 y=313.857 z=-3.219 mm, rx=-0.1302 ry=-1.6605 rz=-0.1403 rad; joints [-65.067, -50.619, 153.092, -93.35, 35.027, 81.724] deg; TCP offset x=0 y=0 z=246 mm, rx=0 ry=0 rz=0 rad
      Waypoint Waypoint_2: TCP in base x=-1013.668 y=283.774 z=13.404 mm, rx=-0.1302 ry=-1.6605 rz=-0.1403 rad; joints [-36.803, -53.188, 133.142, -74.065, 63.057, 86.565] deg
  Wait Sleep waitTime=1
  tp := get_actual_tcp_pose()
  SuppressedNode
    Script file /programs/analyze_touchpoints.script
      | # this file creates the function for analyzing touchpoints
      | # define pi
      | pi = 3.1415926535
      | 
      | # this is the main entry point for calculations.
      | # it takes in the 5 points, analyzes the shape of the box, and then calculates path points and returns them
      | # specifically for Down, Over, then Around (DOtA)
      | # specifically for right-sided boxes (vertical weld on right side of edge)
      | def main_calculate_right(p11, p12, p21, p22, p3, p13, p23, chamferover):
      |     struct1 = analyze_touchpoints_only(p11, p12, p21, p22, p3)
      |     list1 = analyze_vertical_touchpoints(p11, p12, p13, p21, p22, p23, p3)
      |     struct2 = calculate_DOtA_points_right(struct1, list1, chamferover)
      |     validity = check_validity_right(struct1, struct2)
      |     return struct2
      | end
      | 
      | # this is the main entry point for calculations.
      | # it takes in the 5 points, analyzes the shape of the box, and then calculates path points and returns them
      | # specifically for Down, Over, then Around (DOtA)
      | # specifically for left-sided boxes (vertical weld on left side of edge)
      | def main_calculate_left(p11, p12, p21, p22, p3, p13, p23, chamferover):
      |     struct1 = analyze_touchpoints_only(p11, p12, p21, p22, p3)
      |     list1 = analyze_vertical_touchpoints(p11, p12, p13, p21, p22, p23, p3)
      |     struct2 = calculate_DOtA_points_left(struct1, list1, chamferover)
      |     validity = check_validity_left(struct1, struct2)
      |     return struct2
      | end
      | 
      | # this is the main entry point for calculations, for Floor Corner Extended.
      | # it takes in the 7 touchpoints, analyzes the shape of the box.
      | # takes in the user defined point for the top of the weld (tcp_pose_top) and then calculates path points
      | # loopingly tries to calculate the extension along the sidewall that fulfills get_inverse_kin_has_solution() and provides the farthest extension possible
      | # returns the pathpoints
      | # specifically for Down, Over, then Around (DOtA)
      | # specifically for right-sided boxes (vertical weld on right side of edge)
      | def main_calculate_right_extended(p11, p12, p21, p22, p3, p13, p23, chamferover, tcp_pose_top):
      |     struct1 = analyze_touchpoints_only(p11, p12, p21, p22, p3)
      |     list1 = analyze_vertical_touchpoints(p11, p12, p13, p21, p22, p23, p3)
      |     struct2 = calculate_DOtA_points_right_extended(struct1, list1, chamferover, tcp_pose_top)
      |     validity = check_validity_right(struct1, struct2)
      |     return struct2
      | end
      | 
      | # this is the main entry point for calculations, for Floor Corner Extended.
      | # it takes in the 7 touchpoints, analyzes the shape of the box.
      | # takes in the user defined point for the top of the weld (tcp_pose_top) and then calculates path points
      | # loopingly tries to calculate the extension along the sidewall that fulfills get_inverse_kin_has_solution() and provides the farthest extension possible
      | # returns the pathpoints
      | # specifically for Down, Over, then Around (DOtA)
      | # specifically for left-sided boxes (vertical weld on left side of edge)
      | def main_calculate_left_extended(p11, p12, p21, p22, p3, p13, p23, chamferover, tcp_pose_top):
      |     struct1 = analyze_touchpoints_only(p11, p12, p21, p22, p3)
      |     list1 = analyze_vertical_touchpoints(p11, p12, p13, p21, p22, p23, p3)
      |     struct2 = calculate_DOtA_points_left_extended(struct1, list1, chamferover, tcp_pose_top)
      |     validity = check_validity_left(struct1, struct2)
      |     return struct2
      | end
      | 
      | # it takes 5 arguments as points
      | # it returns a struct containing: (pointintersect, pointapproach1, pointapproach2, point1, point2, point3, point4, point5, pointreturn1, heading1, heading2, heading3, path2r1, path2r2, path2l1, path2l2)
      | # specifically for Around then Up (AtU)
      | def analyze_touchpoints(p11, p12, p21, p22, p3):
      |   # FIND THE INTERSECTION
      |   # comment get the z
      |   zcoord=p3[2]
      | 
      |   # get the raw points from the first line
      |   l1p1x=p11[0]
      |   l1p1y=p11[1]
      |   l1p2x=p12[0]
      |   l1p2y=p12[1]
      | 
      |   # equate the first line in 2d space
      |   ml1 = (l1p2y-l1p1y) / (l1p2x-l1p1x)
      | 
      |   # b = y - mx
      |   bl1 = l1p1y - ml1 * l1p1x
      | 
      |   # get the raw points from the second line
      |   l2p1x=p21[0]
      |   l2p1y=p21[1]
      |   l2p2x=p22[0]
      |   l2p2y=p22[1]
      | 
      |   # equate the second line in 2d space
      |   ml2 = (l2p2y-l2p1y) / (l2p2x-l2p1x)
      | 
      |   # b = y - mx
      |   bl2 = l2p1y - ml2 * l2p1x
      | 
      | 
      |   # find the intersection of the two lines
      |   # m1x+b1 = m2x+b2
      |   # m1x - m2x = b2 - b1
      |   # x = (b2-b1) / (m1-m2)
      |   xintersect = (bl2-bl1) / (ml1-ml2)
      |   yintersect = ml1 * xintersect + bl1
      | 
      |   #FIND THE VECTORS
      |   #define a vector from the intersection to the second point on the first line
      |   l1delxfull = l1p2x - xintersect
      |   l1delyfull = l1p2y - yintersect
      | 
      |   l1delmag = sqrt(l1delxfull*l1delxfull + l1delyfull*l1delyfull)
      | 
      |   l1delxunit = l1delxfull / l1delmag
      |   l1delyunit = l1delyfull / l1delmag
      | 
      |   #define a vector from the intersection to the second point on the second line
      |   l2delxfull = l2p2x - xintersect
      |   l2delyfull = l2p2y - yintersect
      | 
      |   l2delmag = sqrt(l2delxfull*l2delxfull + l2delyfull*l2delyfull)
      | 
      |   l2delxunit = l2delxfull / l2delmag
      |   l2delyunit = l2delyfull / l2delmag
      | 
      |   # FIND THE FOUR POINTS ON THE LINES
      |   # find locations 8 inches away from  intersect point
      |   # CONST
      |   welddistance = 8
      |   roundoverdistance = 0.05
      |   zup = .375
      |   # inches
      |   wd = welddistance * 25.4 / 1000
      |   rod = roundoverdistance * 25.4 / 1000
      |   zup = zup * 25.4 / 1000
      | 
      |   # now we have the unit vector. extend the weld distance from the intersection
      |   x = xintersect + l1delxunit * wd
      |   y = yintersect + l1delyunit * wd
      |   z = zcoord + zup
      | 
      |   point1 = p[x,y,z,1.570796,0,0] # dummy orientation for now
      | 
      |   x = xintersect + l1delxunit * rod
      |   y = yintersect + l1delyunit * rod
      | 
      |   point2 = p[x,y,z,1.570796,0,0]
      | 
      |   # now we have the unit vector. extend the weld distance from the intersection
      |   x = xintersect + l2delxunit * wd
      |   y = yintersect + l2delyunit * wd
      | 
      |   point5 = p[x,y,z,0,-1.570796,0]
      | 
      |   x = xintersect + l2delxunit * rod
      |   y = yintersect + l2delyunit * rod
      | 
      |   point4 = p[x,y,z,0,-1.570796,0]
      | 
      |   #DEFINE APPROACH POINTS
      |   pointintersect = p[xintersect,yintersect,zcoord,0,0,0]
      |   pointapproach1 = p[xintersect+0.1,yintersect+0.1,z,1.570796,0,0]
      |   pointapproach2 = p[point1[0], point1[1]+0.1, point1[2], point1[3], point1[4], point1[5]]
      |   pointreturn1 = p[point5[0]+0.1, point5[1], point5[2], point5[3], point5[4], point5[5]]
      | 
      |   #FIND HEADINGS
      |   #for each heading, find the angle of the line with respect to the pos x axis. then add/subtract 90 degrees because you want to be perpendicular to that
      |   headingvector1 = convert_uv_to_heading(l1delxunit, l1delyunit)
      |   headingvector2 = convert_uv_to_heading(l2delxunit, l2delyunit)
      |   # find halfway heading
      |   heading2 = (headingvector1 + headingvector2)/2
      |   # find headings that the robot should face while traveling, perpendicular to the vectors of the sides of the box
      |   heading1 = headingvector1 + pi/2
      |   heading3 = headingvector2 - pi/2
      | 
      |   #FIND POINT 3
      |   #see if we have to / can find point 3
      |   findpoint3 = True
      |   if roundoverdistance == 0:
      |     findpoint3 = False
      |   end
      |   if findpoint3:
      |     # i need to find the point3 such that the arc from p2 to p3 to p4 is tangent to p1-p2 and p4-p5. making this a smooth path will be good
      |     # the direction of movement is from pointintersect in the direction of heading2
      |     # how much movement though? this will depend on whether it is actually a 90 degree angle or not.
      |     # first, find the perpendicular lines through points 2 and 4
      |     perp2 = find_perpendicular_line(ml1, point2[0], point2[1])
      |     perp4 = find_perpendicular_line(ml2, point4[0], point4[1])
      |     # next, find the intersection of those two lines
      |     perpintersect = find_intersection(perp2[0], perp2[1], perp4[0], perp4[1])
      |     radiusofcircle = distance_between(perpintersect[0], perpintersect[1], 0, point2[0], point2[1], 0)
      |     # find a vector the direction of heading2
      |     uvx = cos(heading2)
      |     uvy = sin(heading2)
      |     # compute point3. pass in negative radius because the direction is into the tank but we want to move from the intersection out to the rounded edge
      |     point3coords = add_vectordistance_to_point(perpintersect[0], perpintersect[1], z, uvx, uvy, 0, -1 * radiusofcircle)
      |     point3 = p[point3coords[0], point3coords[1], point3coords[2], 0, 0, 0]
      |   end
      | 
      |   #APPLY ACTUAL RXRYRZ TO POINTS
      |   # convert the headings to rxryrz and insert those values into the relevant points
      |   rxryrz = convert_heading_to_axang(heading1)
      |   rx = rxryrz[0]
      |   ry = rxryrz[1]
      |   rz = rxryrz[2]
      |   pointapproach1 = p[pointapproach1[0], pointapproach1[1], pointapproach1[2], rx, ry, rz]
      |   pointapproach2 = p[pointapproach2[0], pointapproach2[1], pointapproach2[2], rx, ry, rz]
      |   point1 = p[point1[0], point1[1], point1[2], rx, ry, rz]
      |   point2 = p[point2[0], point2[1], point2[2], rx, ry, rz]
      |   rxryrz = convert_heading_to_axang(heading2)
      |   rx = rxryrz[0]
      |   ry = rxryrz[1]
      |   rz = rxryrz[2]
      |   if findpoint3:
      |     point3 = p[point3[0], point3[1], point3[2], rx, ry, rz]
      |   else:
      |     point3 = point2
      |   end
      |   rxryrz = convert_heading_to_axang(heading3)
      |   rx = rxryrz[0]
      |   ry = rxryrz[1]
      |   rz = rxryrz[2]
      |   point4 = p[point4[0], point4[1], point4[2], rx, ry, rz]
      |   point5 = p[point5[0], point5[1], point5[2], rx, ry, rz]
      |   pointreturn1 = p[pointreturn1[0], pointreturn1[1], pointreturn1[2], rx, ry, rz]
      | 
      |   #find path2 (the part that goes up)
      |   four_vertical_points = find_vertical_points(pointintersect, l1delxunit, l1delyunit, l2delxunit, l2delyunit, zup, wd, heading1, heading3)
      |   path2r1 = four_vertical_points[0]
      |   path2r2 = four_vertical_points[1]
      |   path2l1 = four_vertical_points[2]
      |   path2l2 = four_vertical_points[3]
      | 
      |   #RETURN STRUCT
      |   ret = struct(pointintersect=pointintersect, pointapproach1=pointapproach1, pointapproach2=pointapproach2, point1=point1, point2=point2, point3=point3, point4=point4, point5=point5, pointreturn1=pointreturn1, heading1=heading1, heading2=heading2, heading3=heading3, path2r1=path2r1, path2r2=path2r2, path2l1=path2l1, path2l2=path2l2)
      |   return ret
      | end
      | 
      | # it takes 5 arguments as points
      | # it returns a struct containing: (pointintersect, heading1, heading2, heading3, l1delxunit, l1delyunit, l2delxunit, l2delyunit)
      | def analyze_touchpoints_only(p11, p12, p21, p22, p3):
      |   # FIND THE INTERSECTION
      |   # comment get the z
      |   zcoord=p3[2]
      | 
      |   # get the raw points from the first line
      |   l1p1x=p11[0]
      |   l1p1y=p11[1]
      |   l1p2x=p12[0]
      |   l1p2y=p12[1]
      | 
      |   # equate the first line in 2d space
      |   ml1 = (l1p2y-l1p1y) / (l1p2x-l1p1x)
      | 
      |   # b = y - mx
      |   bl1 = l1p1y - ml1 * l1p1x
      | 
      |   # get the raw points from the second line
      |   l2p1x=p21[0]
      |   l2p1y=p21[1]
      |   l2p2x=p22[0]
      |   l2p2y=p22[1]
      | 
      |   # equate the second line in 2d space
      |   ml2 = (l2p2y-l2p1y) / (l2p2x-l2p1x)
      | 
      |   # b = y - mx
      |   bl2 = l2p1y - ml2 * l2p1x
      | 
      | 
      |   # find the intersection of the two lines
      |   # m1x+b1 = m2x+b2
      |   # m1x - m2x = b2 - b1
      |   # x = (b2-b1) / (m1-m2)
      |   xintersect = (bl2-bl1) / (ml1-ml2)
      |   yintersect = ml1 * xintersect + bl1
      | 
      |   pointintersect = p[xintersect,yintersect,zcoord,0,0,0]
      | 
      |   #FIND THE VECTORS
      |   #define a vector from the intersection to the second point on the first line
      |   l1delxfull = l1p2x - xintersect
      |   l1delyfull = l1p2y - yintersect
      | 
      |   l1delmag = sqrt(l1delxfull*l1delxfull + l1delyfull*l1delyfull)
      | 
      |   l1delxunit = l1delxfull / l1delmag
      |   l1delyunit = l1delyfull / l1delmag
      | 
      |   #define a vector from the intersection to the second point on the second line
      |   l2delxfull = l2p2x - xintersect
      |   l2delyfull = l2p2y - yintersect
      | 
      |   l2delmag = sqrt(l2delxfull*l2delxfull + l2delyfull*l2delyfull)
      | 
      |   l2delxunit = l2delxfull / l2delmag
      |   l2delyunit = l2delyfull / l2delmag
      | 
      |   #FIND HEADINGS
      |   #for each heading, find the angle of the line with respect to the pos x axis. then add/subtract 90 degrees because you want to be perpendicular to that
      |   headingvector1 = convert_uv_to_heading(l1delxunit, l1delyunit)
      |   headingvector2 = convert_uv_to_heading(l2delxunit, l2delyunit)
      |   # find halfway heading
      |   heading2 = (headingvector1 + headingvector2)/2
      |   # find headings that the robot should face while traveling, perpendicular to the vectors of the sides of the box
      |   heading1 = headingvector1 + pi/2
      |   heading3 = headingvector2 - pi/2
      | 
      |   #RETURN STRUCT
      |   ret = struct(pointintersect=pointintersect, heading1=heading1, heading2=heading2, heading3=heading3, l1delxunit=l1delxunit, l1delyunit=l1delyunit, l2delxunit=l2delxunit, l2delyunit=l2delyunit)
      |   return ret
      | end
      | 
      | # given a struct from analyze_touchpoints_only(), calculate the points
      | # for right, for non-extended
      | def calculate_DOtA_points_right(struct1, listleans, chamferover):
      |     # get the stuff from the struct
      |     pointintersect = struct1[0]
      |     heading1 = struct1[1]
      |     heading2 = struct1[2]
      |     heading3 = struct1[3]
      |     l1delxunit = struct1[4]
      |     l1delyunit = struct1[5]
      |     l2delxunit = struct1[6]
      |     l2delyunit = struct1[7]
      | 
      |     # FIND THE POINTS ON THE LINES OF THE FIRST TURN PATH
      |     # find locations 8 inches away from  intersect point
      |     # CONST
      |     welddistance1 = 8 # vertical weld distance
      |     welddistance2 = 6 # first path second leg
      |     welddistance3 = 8 # second path second leg
      |     zup = .375
      |     # inches
      |     wd1 = welddistance1 * 25.4 / 1000
      |     wd2 = welddistance2 * 25.4 / 1000
      |     wd3 = welddistance3 * 25.4 / 1000
      |     zup = zup * 25.4 / 1000
      |     chamferovermm =  chamferover * 25.4 / 1000
      | 
      |     x = pointintersect[0] + l1delxunit * chamferovermm
      |     y = pointintersect[1] + l1delyunit * chamferovermm
      |     z = pointintersect[2] + zup
      | 
      |     #apply actual rxryrz to points
      |     # convert the headings to rxryrz and insert those values into the relevant points
      |     rxryrz = convert_heading_to_axang_preheatdown(heading1)
      |     rx = rxryrz[0]
      |     ry = rxryrz[1]
      |     rz = rxryrz[2]
      | 
      |     point1 = p[x + wd1*listleans[0], y + wd1*listleans[1], z + wd1, rx, ry, rz] # add in the listleans factor to follow the face of the box as we move up
      |     point2 = p[x, y, z, rx, ry, rz]
      | 
      |     # convert the headings to rxryrz and insert those values into the relevant points
      |     rxryrz = convert_heading_to_axang_ccw(heading1)
      |     rx = rxryrz[0]
      |     ry = rxryrz[1]
      |     rz = rxryrz[2]
      | 
      |     point4 = p[x, y, z, rx, ry, rz]
      |     x = x + l1delxunit * wd2
      |     y = y + l1delyunit * wd2
      |     point5 = p[x, y, z, rx, ry, rz]
      | 
      |     # FIND THE POINTS ON THE LINES OF THE SECOND AROUND PATH
      |     roundoverdistance = 0.05
      |     rod = roundoverdistance * 25.4 / 1000
      | 
      |     # now we have the unit vector. extend the weld distance from the intersection
      |     x = pointintersect[0] + l1delxunit * chamferovermm
      |     y = pointintersect[1] + l1delyunit * chamferovermm
      |     # convert the headings to rxryrz and insert those values into the relevant points
      |     rxryrz = convert_heading_to_axang(heading1)
      |     rx = rxryrz[0]
      |     ry = rxryrz[1]
      |     rz = rxryrz[2]
      |     point_1 = p[x, y, z, rx, ry, rz]
      | 
      |     x = pointintersect[0] + l1delxunit * rod
      |     y = pointintersect[1] + l1delyunit * rod
      |     point_2 = p[x, y, z, rx, ry, rz]
      | 
      |     # now we have the unit vector. extend the weld distance from the intersection
      |     x = pointintersect[0] + l2delxunit * wd3
      |     y = pointintersect[1] + l2delyunit * wd3
      |     # convert the headings to rxryrz and insert those values into the relevant points
      |     rxryrz = convert_heading_to_axang(heading3)
      |     rx = rxryrz[0]
      |     ry = rxryrz[1]
      |     rz = rxryrz[2]
      |     point_5 = p[x, y, z, rx, ry, rz]
      | 
      |     x = pointintersect[0] + l2delxunit * rod
      |     y = pointintersect[1] + l2delyunit * rod
      |     point_4 = p[x, y, z, rx, ry, rz]
      | 
      |     #FIND POINT 3
      |     # by calling analyze_touchpoints()
      |     atret = analyze_touchpoints(point_2, point_1, point_4, point_5, pointintersect)
      |     point_3 = atret[5]
      | 
      | 
      |     struct2 = struct(point1=point1, point2=point2, point4=point4, point5=point5, point_1=point_1, point_2=point_2, point_3=point_3, point_4=point_4, point_5=point_5)
      |     return struct2
      | end
      | 
      | # given a struct from analyze_touchpoints_only(), calculate the points
      | # for left, for non-extended
      | def calculate_DOtA_points_left(struct1, listleans, chamferover):
      |     # get the stuff from the struct
      |     pointintersect = struct1[0]
      |     heading1 = struct1[1]
      |     heading2 = struct1[2]
      |     heading3 = struct1[3]
      |     l1delxunit = struct1[4]
      |     l1delyunit = struct1[5]
      |     l2delxunit = struct1[6]
      |     l2delyunit = struct1[7]
      | 
      |     # FIND THE POINTS ON THE LINES OF THE FIRST TURN PATH
      |     # find locations 8 inches away from  intersect point
      |     # CONST
      |     welddistance1 = 8 # vertical weld distance
      |     welddistance2 = 6 # first path second leg
      |     welddistance3 = 8 # second path second leg
      |     zup = .375
      |     # inches
      |     wd1 = welddistance1 * 25.4 / 1000
      |     wd2 = welddistance2 * 25.4 / 1000
      |     wd3 = welddistance3 * 25.4 / 1000
      |     zup = zup * 25.4 / 1000
      |     chamferovermm =  chamferover * 25.4 / 1000
      | 
      |     x = pointintersect[0] + l2delxunit * chamferovermm
      |     y = pointintersect[1] + l2delyunit * chamferovermm
      |     z = pointintersect[2] + zup
      | 
      |     #apply actual rxryrz to points
      |     # convert the headings to rxryrz and insert those values into the relevant points
      |     rxryrz = convert_heading_to_axang_preheatdown(heading3)
      |     rx = rxryrz[0]
      |     ry = rxryrz[1]
      |     rz = rxryrz[2]
      | 
      |     point1 = p[x + wd1*listleans[0], y + wd1*listleans[1], z + wd1, rx, ry, rz]
      |     point2 = p[x, y, z, rx, ry, rz]
      | 
      |     # convert the headings to rxryrz and insert those values into the relevant points
      |     rxryrz = convert_heading_to_axang(heading3)
      |     rx = rxryrz[0]
      |     ry = rxryrz[1]
      |     rz = rxryrz[2]
      | 
      |     point4 = p[x, y, z, rx, ry, rz]
      |     x = x + l2delxunit * wd2
      |     y = y + l2delyunit * wd2
      |     point5 = p[x, y, z, rx, ry, rz]
      | 
      |     # FIND THE POINTS ON THE LINES OF THE SECOND AROUND PATH
      |     roundoverdistance = 0.05
      |     rod = roundoverdistance * 25.4 / 1000
      | 
      |     # now we have the unit vector. extend the weld distance from the intersection
      |     x = pointintersect[0] + l2delxunit * chamferovermm
      |     y = pointintersect[1] + l2delyunit * chamferovermm
      |     # convert the headings to rxryrz and insert those values into the relevant points
      |     rxryrz = convert_heading_to_axang_ccw(heading3)
      |     rx = rxryrz[0]
      |     ry = rxryrz[1]
      |     rz = rxryrz[2]
      |     point_1 = p[x, y, z, rx, ry, rz]
      | 
      |     x = pointintersect[0] + l2delxunit * rod
      |     y = pointintersect[1] + l2delyunit * rod
      |     point_2 = p[x, y, z, rx, ry, rz]
      | 
      |     # now we have the unit vector. extend the weld distance from the intersection
      |     x = pointintersect[0] + l1delxunit * wd3
      |     y = pointintersect[1] + l1delyunit * wd3
      |     # convert the headings to rxryrz and insert those values into the relevant points
      |     rxryrz = convert_heading_to_axang_ccw(heading1)
      |     rx = rxryrz[0]
      |     ry = rxryrz[1]
      |     rz = rxryrz[2]
      |     point_5 = p[x, y, z, rx, ry, rz]
      | 
      |     x = pointintersect[0] + l1delxunit * rod
      |     y = pointintersect[1] + l1delyunit * rod
      |     point_4 = p[x, y, z, rx, ry, rz]
      | 
      |     #FIND POINT 3
      |     # by calling analyze_touchpoints()
      |     atret = analyze_touchpoints(point_2, point_1, point_4, point_5, pointintersect)
      |     point_3 = atret[5]
      |     #point 3 will not have the correct rxryrz though because now the gun needs to be face up.
      |     rxryrz = convert_heading_to_axang_ccw(heading2)
      |     rx = rxryrz[0]
      |     ry = rxryrz[1]
      |     rz = rxryrz[2]
      |     point_3 = p[point_3[0], point_3[1], point_3[2], rx, ry, rz]
      | 
      |     struct2 = struct(point1=point1, point2=point2, point4=point4, point5=point5, point_1=point_1, point_2=point_2, point_3=point_3, point_4=point_4, point_5=point_5)
      |     return struct2
      | end
      | 
      | # given a struct from analyze_touchpoints_only(), calculate the points
      | # for right, for extended
      | def calculate_DOtA_points_right_extended(struct1, listleans, chamferover, tcp_pose_top):
      |     # get the stuff from the struct
      |     pointintersect = struct1[0]
      |     heading1 = struct1[1]
      |     heading2 = struct1[2]
      |     heading3 = struct1[3]
      |     l1delxunit = struct1[4]
      |     l1delyunit = struct1[5]
      |     l2delxunit = struct1[6]
      |     l2delyunit = struct1[7]
      | 
      |     # FIND THE POINTS ON THE LINES OF THE FIRST TURN PATH
      |     # find locations 8 inches away from  intersect point
      |     # CONST
      |     # welddistance1 = 8 # vertical weld distance
      |     welddistance2 = 6 # first path second leg
      |     welddistance3 = 8 # second path second leg
      |     zup = .375
      |     # inches
      |     # wd1 = welddistance1 * 25.4 / 1000
      |     wd2 = welddistance2 * 25.4 / 1000
      |     wd3 = welddistance3 * 25.4 / 1000
      |     zup = zup * 25.4 / 1000
      |     chamferovermm =  chamferover * 25.4 / 1000
      | 
      |     # weld distance is the distance that it will weld. this will make it start at the z height that the user specified
      |     wd1 = tcp_pose_top[2] - pointintersect[2] - zup
      | 
      |     x = pointintersect[0] + l1delxunit * chamferovermm
      |     y = pointintersect[1] + l1delyunit * chamferovermm
      |     z = pointintersect[2] + zup
      | 
      |     #apply actual rxryrz to points
      |     # convert the headings to rxryrz and insert those values into the relevant points
      |     rxryrz = convert_heading_to_axang_preheatdown(heading1)
      |     rx = rxryrz[0]
      |     ry = rxryrz[1]
      |     rz = rxryrz[2]
      | 
      |     point1 = p[x + wd1*listleans[0], y + wd1*listleans[1], z + wd1, rx, ry, rz] # add in the listleans factor to follow the face of the box as we move up
      |     point2 = p[x, y, z, rx, ry, rz]
      | 
      |     # convert the headings to rxryrz and insert those values into the relevant points
      |     rxryrz = convert_heading_to_axang_ccw(heading1)
      |     rx = rxryrz[0]
      |     ry = rxryrz[1]
      |     rz = rxryrz[2]
      | 
      |     point4 = p[x, y, z, rx, ry, rz]
      |     x = x + l1delxunit * wd2
      |     y = y + l1delyunit * wd2
      |     point5 = p[x, y, z, rx, ry, rz]
      | 
      |     # FIND THE POINTS ON THE LINES OF THE SECOND AROUND PATH
      |     roundoverdistance = 0.05
      |     rod = roundoverdistance * 25.4 / 1000
      | 
      |     # now we have the unit vector. extend the weld distance from the intersection
      |     x = pointintersect[0] + l1delxunit * chamferovermm
      |     y = pointintersect[1] + l1delyunit * chamferovermm
      |     # convert the headings to rxryrz and insert those values into the relevant points
      |     rxryrz = convert_heading_to_axang(heading1)
      |     rx = rxryrz[0]
      |     ry = rxryrz[1]
      |     rz = rxryrz[2]
      |     point_1 = p[x, y, z, rx, ry, rz]
      | 
      |     x = pointintersect[0] + l1delxunit * rod
      |     y = pointintersect[1] + l1delyunit * rod
      |     point_2 = p[x, y, z, rx, ry, rz]
      | 
      |     # convert the headings to rxryrz and insert those values into the relevant points
      |     rxryrz = convert_heading_to_axang(heading3)
      |     rx = rxryrz[0]
      |     ry = rxryrz[1]
      |     rz = rxryrz[2]
      | 
      |     x = pointintersect[0] + l2delxunit * rod
      |     y = pointintersect[1] + l2delyunit * rod
      |     point_4 = p[x, y, z, rx, ry, rz]
      | 
      |     # extend the weld distance from the intersection
      |     valid1 = True
      |     # start with the seed
      |     x = pointintersect[0] + l2delxunit * wd3
      |     y = pointintersect[1] + l2delyunit * wd3
      |     point_5 = p[x, y, z, rx, ry, rz]
      |     seed = p[x, y, z, rx, ry, rz]
      |     valid1 = get_inverse_kin_has_solution(seed)
      |     # define the increment
      |     increment = 1.0 # inches
      |     increment = increment * 25.4 / 1000 # meters
      |     while valid1 == True:
      |         wd3 = wd3 + increment
      |         x = pointintersect[0] + l2delxunit * wd3
      |         y = pointintersect[1] + l2delyunit * wd3
      |         seed = p[x, y, z, rx, ry, rz]
      |         valid1 = get_inverse_kin_has_solution(seed)
      |     end
      |     # move back 1 to get the highest valid wd3
      |     # move back 3 to get the third highest valid wd3
      |     wd3 = wd3 - (3.0 * increment)
      |     x = pointintersect[0] + l2delxunit * wd3
      |     y = pointintersect[1] + l2delyunit * wd3
      |     point_5 = p[x, y, z, rx, ry, rz]
      | 
      |     #FIND POINT 3
      |     # by calling analyze_touchpoints()
      |     atret = analyze_touchpoints(point_2, point_1, point_4, point_5, pointintersect)
      |     point_3 = atret[5]
      | 
      | 
      |     struct2 = struct(point1=point1, point2=point2, point4=point4, point5=point5, point_1=point_1, point_2=point_2, point_3=point_3, point_4=point_4, point_5=point_5)
      |     return struct2
      | end
      | 
      | # given a struct from analyze_touchpoints_only(), calculate the points
      | # for left, for extended
      | def calculate_DOtA_points_left_extended(struct1, listleans, chamferover, tcp_pose_top):
      |     # get the stuff from the struct
      |     pointintersect = struct1[0]
      |     heading1 = struct1[1]
      |     heading2 = struct1[2]
      |     heading3 = struct1[3]
      |     l1delxunit = struct1[4]
      |     l1delyunit = struct1[5]
      |     l2delxunit = struct1[6]
      |     l2delyunit = struct1[7]
      | 
      |     # FIND THE POINTS ON THE LINES OF THE FIRST TURN PATH
      |     # find locations 8 inches away from  intersect point
      |     # CONST
      |     # welddistance1 = 8 # vertical weld distance
      |     welddistance2 = 6 # first path second leg
      |     welddistance3 = 8 # second path second leg
      |     zup = .375
      |     # inches
      |     # wd1 = welddistance1 * 25.4 / 1000
      |     wd2 = welddistance2 * 25.4 / 1000
      |     wd3 = welddistance3 * 25.4 / 1000
      |     zup = zup * 25.4 / 1000
      |     chamferovermm =  chamferover * 25.4 / 1000
      | 
      |     # weld distance is the distance that it will weld. this will make it start at the z height that the user specified
      |     wd1 = tcp_pose_top[2] - pointintersect[2] - zup
      | 
      |     x = pointintersect[0] + l2delxunit * chamferovermm
      |     y = pointintersect[1] + l2delyunit * chamferovermm
      |     z = pointintersect[2] + zup
      | 
      |     #apply actual rxryrz to points
      |     # convert the headings to rxryrz and insert those values into the relevant points
      |     rxryrz = convert_heading_to_axang_preheatdown(heading3)
      |     rx = rxryrz[0]
      |     ry = rxryrz[1]
      |     rz = rxryrz[2]
      | 
      |     point1 = p[x + wd1*listleans[0], y + wd1*listleans[1], z + wd1, rx, ry, rz]
      |     point2 = p[x, y, z, rx, ry, rz]
      | 
      |     # convert the headings to rxryrz and insert those values into the relevant points
      |     rxryrz = convert_heading_to_axang(heading3)
      |     rx = rxryrz[0]
      |     ry = rxryrz[1]
      |     rz = rxryrz[2]
      | 
      |     point4 = p[x, y, z, rx, ry, rz]
      |     x = x + l2delxunit * wd2
      |     y = y + l2delyunit * wd2
      |     point5 = p[x, y, z, rx, ry, rz]
      | 
      |     # FIND THE POINTS ON THE LINES OF THE SECOND AROUND PATH
      |     roundoverdistance = 0.05
      |     rod = roundoverdistance * 25.4 / 1000
      | 
      |     # now we have the unit vector. extend the weld distance from the intersection
      |     x = pointintersect[0] + l2delxunit * chamferovermm
      |     y = pointintersect[1] + l2delyunit * chamferovermm
      |     # convert the headings to rxryrz and insert those values into the relevant points
      |     rxryrz = convert_heading_to_axang_ccw(heading3)
      |     rx = rxryrz[0]
      |     ry = rxryrz[1]
      |     rz = rxryrz[2]
      |     point_1 = p[x, y, z, rx, ry, rz]
      | 
      |     x = pointintersect[0] + l2delxunit * rod
      |     y = pointintersect[1] + l2delyunit * rod
      |     point_2 = p[x, y, z, rx, ry, rz]
      | 
      |     # convert the headings to rxryrz and insert those values into the relevant points
      |     rxryrz = convert_heading_to_axang_ccw(heading1)
      |     rx = rxryrz[0]
      |     ry = rxryrz[1]
      |     rz = rxryrz[2]
      | 
      |     x = pointintersect[0] + l1delxunit * rod
      |     y = pointintersect[1] + l1delyunit * rod
      |     point_4 = p[x, y, z, rx, ry, rz]
      | 
      |     # extend the weld distance from the intersection
      |     valid1 = True
      |     # start with the seed
      |     x = pointintersect[0] + l1delxunit * wd3
      |     y = pointintersect[1] + l1delyunit * wd3
      |     point_5 = p[x, y, z, rx, ry, rz]
      |     seed = p[x, y, z, rx, ry, rz]
      |     valid1 = get_inverse_kin_has_solution(seed)
      |     # define the increment
      |     increment = 1.0 # inches
      |     increment = increment * 25.4 / 1000 # meters
      |     while valid1 == True:
      |         wd3 = wd3 + increment
      |         x = pointintersect[0] + l1delxunit * wd3
      |         y = pointintersect[1] + l1delyunit * wd3
      |         seed = p[x, y, z, rx, ry, rz]
      |         valid1 = get_inverse_kin_has_solution(seed)
      |     end
      |     # move back 1 to get the highest valid wd3
      |     # move back 3 to get the third highest valid wd3
      |     wd3 = wd3 - (3.0 * increment)
      |     x = pointintersect[0] + l1delxunit * wd3
      |     y = pointintersect[1] + l1delyunit * wd3
      |     point_5 = p[x, y, z, rx, ry, rz]
      | 
      |     #FIND POINT 3
      |     # by calling analyze_touchpoints()
      |     atret = analyze_touchpoints(point_2, point_1, point_4, point_5, pointintersect)
      |     point_3 = atret[5]
      |     #point 3 will not have the correct rxryrz though because now the gun needs to be face up
      |     rxryrz = convert_heading_to_axang_ccw(heading2)
      |     rx = rxryrz[0]
      |     ry = rxryrz[1]
      |     rz = rxryrz[2]
      |     point_3 = p[point_3[0], point_3[1], point_3[2], rx, ry, rz]
      | 
      |     struct2 = struct(point1=point1, point2=point2, point4=point4, point5=point5, point_1=point_1, point_2=point_2, point_3=point_3, point_4=point_4, point_5=point_5)
      |     return struct2
      | end
      | 
      | # this function analyzes the vertical points
      | # calculates the slope of the edge in question
      | # specifically, for each inch up in the z direction, what is the change in x and change in y direction
      | # returns a list of [nx, ny]
      | def analyze_vertical_touchpoints(p11, p12, p13, p21, p22, p23, p3):
      |     # first, find the equations of the planes from the 6 points
      |     plane1 = findplane(p11, p12, p13)
      |     plane2 = findplane(p21, p22, p23)
      |     # Find the Direction Vector of the Line: The direction vector d of the line of intersection can be found by taking the cross product of the normal vectors of each plane (a, b, and c)
      |     nx = plane1[1]*plane2[2] - plane1[2]*plane2[1]
      |     ny = plane1[2]*plane2[0] - plane1[0]*plane2[2]
      |     nz = plane1[0]*plane2[1] - plane1[1]*plane2[0]
      |     # normalize the vector so the z length is 1
      |     multiplier = 1 / nz
      |     nx = nx * multiplier
      |     ny = ny * multiplier
      |     nz = nz * multiplier # should become equal to 1
      |     ret = [nx, ny]
      |     return ret
      | end
      | 
      | # given 3 points, this finds the plane and its equation
      | # rereturns ax + by + cz + d = 0 in a list of [a, b, c, d]
      | def findplane(p11, p12, p13):
      |     # extract coordinates
      |     x1 = p11[0]
      |     y1 = p11[1]
      |     z1 = p11[2]
      |     x2 = p12[0]
      |     y2 = p12[1]
      |     z2 = p12[2]
      |     x3 = p13[0]
      |     y3 = p13[1]
      |     z3 = p13[2]
      |     # create vectors from the points
      |     v1x = x2-x1
      |     v1y = y2-y1
      |     v1z = z2-z1
      |     v2x = x3-x1
      |     v2y = y3-y1
      |     v2z = z3-z1
      |     #calculate the normal vector using the cross product
      |     nx = v1y*v2z - v1z*v2y # i component
      |     ny = v1z*v2x - v1x*v2z # j component
      |     nz = v1x*v2y - v1y*v2x # k component
      |     # calculate d in the plane equation
      |     d = -1 * (nx*x1 + ny*y1 + nz*z1)
      |     ret = [nx, ny, nz, d]
      |     return ret
      | end
      | 
      | # given a heading, (ccw from +x axis), find the mx+b slope
      | # fails if exactly vertical
      | def get_slope_from_heading(heading):
      |     return tan(heading)
      | end
      | 
      | 
      | 
      | # this function finds the points (and rxryrz) of the 2 points (start and end) of vertical weld section
      | def find_vertical_points(pointintersect, l1delxunit, l1delyunit, l2delxunit, l2delyunit, offset, wd, heading1, heading3):
      | 
      |   # find right side stuff
      |   # find the point in 3d space that is .375 up and .375 over
      |   x = pointintersect[0] + l1delxunit * offset
      |   y = pointintersect[1] + l1delyunit * offset
      |   z = pointintersect[2] + offset
      |   # find rxryrz
      |   rxryrz = convert_heading_to_axang_preheatup(heading1)
      |   rx = rxryrz[0]
      |   ry = rxryrz[1]
      |   rz = rxryrz[2]
      |   path2r1 = p[x, y, z, rx, ry, rz]
      |   path2r2 = p[x, y, z + wd, rx, ry, rz]
      | 
      |   # find left side
      |   # find the point in 3d space that is .375 up and .375 over
      |   x = pointintersect[0] + l2delxunit * offset
      |   y = pointintersect[1] + l2delyunit * offset
      |   z = pointintersect[2] + offset
      |   # find rxryrz
      |   rxryrz = convert_heading_to_axang_preheatup(heading3)
      |   rx = rxryrz[0]
      |   ry = rxryrz[1]
      |   rz = rxryrz[2]
      |   path2l1 = p[x, y, z, rx, ry, rz]
      |   path2l2 = p[x, y, z + wd, rx, ry, rz]
      | 
      |   ret = struct(path2r1=path2r1, path2r2=path2r2, path2l1=path2l1, path2l2=path2l2)
      |   return ret
      | end
      | 
      | # this function converts a unit vector to its heading angle ccw from x+ axis
      | # takes uvx and uvy
      | # returns heading in radians
      | def convert_uv_to_heading(uvx, uvy):
      |   baseang = atan(uvy/uvx)
      |   if uvx < 0:
      |     ang = baseang + pi
      |   elif uvy < 0:
      |     ang = baseang + pi * 2
      |   else:
      |     ang = baseang
      |   end
      |   return ang
      | end
      | 
      | # this function finds the equation of a line, perpendicular to a given line, and going through a given point
      | # takes 3 arguments: m (the original line's slope), x (point's x coord), y (point's y coord). the b of the original line is not needed
      | # returns a list of [m,b] (the slope and intercept of the new line)
      | def find_perpendicular_line(origm, x, y):
      |   m = (1/origm) * -1
      |   b = y - m*x
      |   ret = [m, b]
      |   return ret
      | end
      | 
      | # this function finds the intersection point between two lines in the xy plane
      | # takes 4 arguments: m1, b1, m2, b2
      | # returns a list of [x,y] (the point of intersection)
      | def find_intersection(m1, b1, m2, b2):
      |   # m1x+b1 = m2x+b2
      |   # m1x - m2x = b2 - b1
      |   # x = (b2-b1) / (m1-m2)
      |   x = (b2-b1) / (m1-m2)
      |   y = m1 * x + b1
      |   ret = [x, y]
      |   return ret
      | end
      | 
      | # this function finds the distance between 2 points in 3d space
      | # it takes 6 arguments: x1, y1, z1, x2, y2, z2
      | # it returns a distance
      | def distance_between(x1, y1, z1, x2, y2, z2):
      |   distsquared = (x2-x1)*(x2-x1)+(y2-y1)*(y2-y1)+(z2-z1)*(z2-z1)
      |   dist = sqrt(distsquared)
      |   return dist
      | end
      | 
      | # this function takes a point, a unit vector, and a distance, and adds the distance to the point in the direction of the unit vector (3d space)
      | # it returns a point as a list of coordinates
      | def add_vectordistance_to_point(xi, yi, zi, uvx, uvy, uvz, delta):
      |   xf = xi + uvx * delta
      |   yf = yi + uvy * delta
      |   zf = zi + uvz * delta
      |   ret = [xf, yf, zf]
      |   return ret
      | end
      | 
      | # this function converts a heading (ccw radians from the positive x axis) into rxryrz to be put into a point p[]
      | # this will point the gun in this heading with the bottom side of the gun facing up.
      | # the values used in this program were calculated by doing rotation matrix math in the file on WI-CALVINB10 C. Documents. Theory for converting rotations into axis angle representations
      | def convert_heading_to_axang(heading):
      |  axisxraw = -1 * sin(heading)
      |  axisyraw = cos(heading) + 1
      |  axiszraw = sin(heading)
      | 
      |  magnitude = sqrt(axisxraw*axisxraw + axisyraw*axisyraw + axiszraw*axiszraw)
      | 
      |  axisxunit = axisxraw / magnitude
      |  axisyunit = axisyraw / magnitude
      |  axiszunit = axiszraw / magnitude
      | 
      |  angle = acos( (cos(heading) - 1) / 2 )
      | 
      |  rxout = axisxunit * angle
      |  ryout = axisyunit * angle
      |  rzout = axiszunit * angle
      | 
      |  return [rxout, ryout, rzout]
      | end
      | 
      | # this function converts a heading (ccw radians from the positive x axis) into rxryrz to be put into a point p[]
      | # this will point the gun in this heading with the preheat side of the gun tip facing up. Used for welding in a vertical path.
      | # the values used in this program were calculated by doing rotation matrix math in the file on WI-CALVINB10 C. Documents. Theory for converting rotations into axis angle representations
      | def convert_heading_to_axang_preheatup(heading):
      |  axisxraw = -sin(heading) + 1
      |  axisyraw = cos(heading)
      |  axiszraw = cos(heading)
      | 
      |  magnitude = sqrt(axisxraw*axisxraw + axisyraw*axisyraw + axiszraw*axiszraw)
      | 
      |  axisxunit = axisxraw / magnitude
      |  axisyunit = axisyraw / magnitude
      |  axiszunit = axiszraw / magnitude
      | 
      |  angle = acos( (-sin(heading) - 1) / 2 )
      | 
      |  rxout = axisxunit * angle
      |  ryout = axisyunit * angle
      |  rzout = axiszunit * angle
      | 
      |  return [rxout, ryout, rzout]
      | end
      | 
      | # this function converts a heading (ccw radians from the positive x axis) into rxryrz to be put into a point p[]
      | # this will point the gun in this heading with the preheat side of the gun tip facing down. Used for welding in a vertical path downwards.
      | # the values used in this program were calculated by doing rotation matrix math in the file on WI-CALVINB10 C. Documents. Theory for converting rotations into axis angle representations
      | def convert_heading_to_axang_preheatdown(heading):
      |  axisxraw = -sin(heading) - 1
      |  axisyraw = cos(heading)
      |  axiszraw = -cos(heading)
      | 
      |  magnitude = sqrt(axisxraw*axisxraw + axisyraw*axisyraw + axiszraw*axiszraw)
      | 
      |  axisxunit = axisxraw / magnitude
      |  axisyunit = axisyraw / magnitude
      |  axiszunit = axiszraw / magnitude
      | 
      |  angle = acos( (sin(heading) - 1) / 2 )
      | 
      |  rxout = axisxunit * angle
      |  ryout = axisyunit * angle
      |  rzout = axiszunit * angle
      | 
      |  return [rxout, ryout, rzout]
      | end
      | 
      | # this function converts a heading (ccw radians from the positive x axis) into rxryrz to be put into a point p[]
      | # this will point the gun in this heading with the preheat side of the gun tip facing right. Used for welding counterclockwise around the box.
      | # the values used in this program were calculated by doing rotation matrix math in the file on WI-CALVINB10 C. Documents. Theory for converting rotations into axis angle representations
      | def convert_heading_to_axang_ccw(heading):
      |  axisxraw = -sin(heading)
      |  axisyraw = cos(heading) - 1
      |  axiszraw = -sin(heading)
      | 
      |  magnitude = sqrt(axisxraw*axisxraw + axisyraw*axisyraw + axiszraw*axiszraw)
      | 
      |  axisxunit = axisxraw / magnitude
      |  axisyunit = axisyraw / magnitude
      |  axiszunit = axiszraw / magnitude
      | 
      |  angle = acos( (-cos(heading) - 1) / 2 )
      | 
      |  rxout = axisxunit * angle
      |  ryout = axisyunit * angle
      |  rzout = axiszunit * angle
      | 
      |  return [rxout, ryout, rzout]
      | end
      | 
      | # this function is for getting the points along the path of the corner homing 45
      | # point0 is the point where they touched
      | def get_corner_homing_45_pathpoints(point0):
      |   p0x = point0[0]
      |   p0y = point0[1]
      |   p0z = point0[2]
      |   p0rx = point0[3]
      |   p0ry = point0[4]
      |   p0rz = point0[5]
      | 
      |   #constants
      |   #distances of how far away from point the touchpoints are
      |   d0 = 0.10 # how far from the box to retreat and approach
      |   d1 = 0.03 # first distance from init point
      |   d2 = 0.15 # second distance from init point
      |   d3 = 0.125 #vertical distance from first point
      |   sqrt2 = 0.707106781 # 1/sqrt(2) , the inverse of the sqrt(2)
      | 
      |   ph1 = p[p0x + d0, p0y, p0z + d1, p0rx, p0ry, p0rz] #approach point for turn
      | 
      |   ph2 = p[p0x+d0-d0*0.5-sqrt2*d1, p0y+d0*0.5+sqrt2*d1, p0z+d1, 1.446, -0.8, -0.733]
      |   ph3 = p[p0x+d0-d0*0.5-sqrt2*d2, p0y+d0*0.5+sqrt2*d2, p0z+d1, 1.446, -0.8, -0.733]
      |   ph4 = p[p0x+d0-d0*0.5-sqrt2*d1, p0y-d0*0.5-sqrt2*d1, p0z+d1, 0.626, -1.993, -1.813]
      |   ph5 = p[p0x+d0-d0*0.5-sqrt2*d2, p0y-d0*0.5-sqrt2*d2, p0z+d1, 0.626, -1.993, -1.813]
      | 
      |   # go back to ph1
      |   ph6 = p[p0x + d0, p0y, p0z -0.05, 0, 0, 0] # approach point for under turn
      |   # moveL from ph1 to ph6
      |   ph7 = p[p0x-d1, p0y, p0z-0.05, 0, 0, 0]
      | 
      |   # add the vertical touch points
      |   ph2up = p[ph2[0], ph2[1], ph2[2]+d3, ph2[3], ph2[4], ph2[5]]
      |   ph4up = p[ph4[0], ph4[1], ph4[2]+d3, ph4[3], ph4[4], ph4[5]]
      |   ret = struct(ph1=ph1, ph2=ph2, ph3=ph3, ph4=ph4, ph5=ph5, ph6=ph6, ph7=ph7, ph2up=ph2up, ph4up=ph4up)
      |   is_robot_at_reachable_spot(point0, ret)
      |   return ret
      | end
      | 
      | # this function checks whether the touchpoints are reachable AKA is the robot positioned in the right spot
      | # if everything looks good, it continues.
      | # if it detects a problem, it infinite loops a popup
      | def is_robot_at_reachable_spot(point0, struct_touchpoints):
      |   # first, check whether the corner is too low to the ground that the bottom homing will hit the ground (z < -350)
      |   if point0[2] < -0.350:
      |     # bad
      |     popuptext = "Tank Corner is too low to the ground. Collisions will occur. Stop Program and raise tank. "
      |     # infinite loop
      |     while 1==1:
      |       popup(popuptext, title="Robot Positioning Warning",blocking=True)
      |     end
      |   end
      | 
      | 
      | 
      |   # next, check whether the touchpoints are reachable
      |   structlength = 9
      |   i = 0
      |   allvalid = True
      |   listproblems = ""
      |   listnames = ["ph1", "ph2", "ph3", "ph4", "ph5", "ph6", "ph7", "ph2up", "ph4up"]
      |   while i < structlength:
      |     curr = struct_touchpoints[i]
      |     valid = get_inverse_kin_has_solution(curr)
      |     if not valid:
      |       allvalid = False
      |       listproblems = listproblems + listnames[i]
      |     end
      |     i = i + 1
      |   end
      | 
      |   if not allvalid:
      |     # display
      |     popuptext = "Robot is too far from tank corner. Cannot reach some necessary positions. Stop Program and move robot closer. " + listproblems
      |     # infinite loop
      |     while 1==1:
      |       popup(popuptext, title="Robot Positioning Warning",blocking=True)
      |     end
      |   end
      | 
      | end
      | 
      | # checks the validity of all points during a left weld
      | def check_validity_left(struct1, struct2):
      |   #first, check whether robot is too close
      |   pointintersect = struct1[0]
      |   # next, check if the corner is too close to the robot to do a left around weld (complex but approximately X > -1300)
      |   # if y < 0, then x < -1300. if y < 480, then y > (1300+x)*8. if y > 480, then y > (1235+x)*4 + 500
      |   toocloseleftweld = False
      |   if pointintersect[1] < 0:
      |     if pointintersect[0] > -1.300:
      |       toocloseleftweld = True
      |     end
      |   elif pointintersect[1] < 0.480:
      |     if pointintersect[1] < (1.300 + pointintersect[0])*8:
      |       toocloseleftweld = True
      |     end
      |   else:
      |     if pointintersect[1] < (1.235 + pointintersect[0])*4 + 0.500:
      |       toocloseleftweld = True
      |     end
      |   end
      |   if toocloseleftweld:
      |     # bad
      |     popuptext = "Robot is too close to tank corner. Collisions may occur. Stop Program and move robot farther. "
      |     # infinite loop
      |     while 1==1:
      |       popup(popuptext, title="Robot Positioning Warning",blocking=True)
      |     end
      |   end
      | 
      |   #next, check whether all the points in the weldpath are valid
      |   structlength = 9
      |   i = 0
      |   allvalid = True
      |   listproblems = ""
      |   listnames = ["point1", "point2", "point4", "point5", "point_1", "point_2", "point_3", "point_4", "point_5"]
      |   while i < structlength:
      |     curr = struct2[i]
      |     valid = get_inverse_kin_has_solution(curr)
      |     if not valid:
      |       allvalid = False
      |       listproblems = listproblems + listnames[i]
      |     end
      |     i = i + 1
      |   end
      | 
      |   if not allvalid:
      |     # display
      |     popuptext = "Robot is too far from tank corner. Cannot reach some necessary positions. Stop Program and move robot closer. " + listproblems
      |     # infinite loop
      |     while 1==1:
      |       popup(popuptext, title="Robot Positioning Warning",blocking=True)
      |     end
      |   end
      | 
      | 
      | end
      | 
      | # checks the validity of all points during a right weld
      | def check_validity_right(struct1, struct2):
      |   # first, check whether the right pivot will bonk itself
      |   pointintersect = struct1[0]
      |   heading1 = struct1[1] # this is the direction that the welder will face when doing the right side of the box
      | 
      |   #first, check whether the heading is just too far offset
      |   # more than 15 degrees off of 45 is too much
      |   # normal heading is 216 degrees
      |   #201 degrees to 231 degrees
      |   heading1degrees = heading1 * 180 / pi
      |   if heading1degrees < 201 or heading1degrees > 231 :
      |     # then out of range
      |     popuptext = "Robot is not aligned at a 45 degree angle of corner (15 degree leeway). Collisions may occur. Stop Program and align robot. heading1degrees=" + str_cat("",heading1degrees)
      |     # infinite loop
      |     while 1==1:
      |       popup(popuptext, title="Robot Positioning Warning",blocking=True)
      |     end
      |   end
      | 
      |   #TODO: add the checks for whether x is too close, given the heading
      |   # add checks for whether x is too close, given the heading
      |   # different equations for whether heading offset > 5 degrees or less (inc. negative)
      |   headingoffset = heading1degrees - 216
      |   if headingoffset < 5:
      |     # then calculate a and b
      |     a = 0.4584 + -0.02369 * headingoffset
      |     b = (-1151.4 + 13.83 * headingoffset) / 1000
      |     # check whether x > a*y+b
      |     if pointintersect[0] > a * pointintersect[1] + b:
      |       # bad
      |       popuptext = "Robot is too close to tank corner or not at the right angle. Collisions may occur. Stop Program and align robot. "
      |       # infinite loop
      |       while 1==1:
      |         popup(popuptext, title="Robot Positioning Warning",blocking=True)
      |       end
      |     end
      |   else:
      |     # headingoffset > 5 degrees
      |     if pointintersect[1] < 0:
      |       if pointintersect[0] > -1150.0 / 1000.0:
      |         #bad
      |         popuptext = "Robot is too close to tank corner. Collisions may occur. Stop Program and align robot. "
      |         # infinite loop
      |         while 1==1:
      |           popup(popuptext, title="Robot Positioning Warning",blocking=True)
      |         end
      |       end
      |     else:
      |       # if x > .7736 y - 1101.9 then bad
      |       if pointintersect[0] > 0.7736 * pointintersect[1] - 1101.9 / 1000:
      |         popuptext = "Robot is too close to tank corner. Collisions may occur. Stop Program and align robot. "
      |         # infinite loop
      |         while 1==1:
      |           popup(popuptext, title="Robot Positioning Warning",blocking=True)
      |         end
      |       end
      |     end
      |   end
      | 
      |   #next, check whether all the points in the weldpath are valid
      |   structlength = 9
      |   i = 0
      |   allvalid = True
      |   listproblems = ""
      |   listnames = ["point1", "point2", "point4", "point5", "point_1", "point_2", "point_3", "point_4", "point_5"]
      |   while i < structlength:
      |     curr = struct2[i]
      |     valid = get_inverse_kin_has_solution(curr)
      |     if not valid:
      |       allvalid = False
      |       listproblems = listproblems + listnames[i]
      |     end
      |     i = i + 1
      |   end
      | 
      |   if not allvalid:
      |     # display
      |     popuptext = "Robot is too far from tank corner. Cannot reach some necessary positions. Stop Program and move robot closer. " + listproblems
      |     # infinite loop
      |     while 1==1:
      |       popup(popuptext, title="Robot Positioning Warning",blocking=True)
      |     end
      |   end
      | end
      | 
      | # this function sends a signal to turn extrusion on
      | def turn_extrusion_on():
      |   # flush the channel
      |   resp0 = send_serial_signal(["u", "r", "?"])
      |   # send the signal
      |   resp1 = send_serial_signal(["u", "R", "1"])
      |   # if resp <> "uR1"
      |   if resp1 != [252,82,49]:
      |     # turn off extrusion and heating. inform calvin
      |     resp2 = send_serial_signal(["u", "R", "0"])
      |     resp3 = send_serial_signal(["u", "H", "0"])
      |     popuptext = "Error code encountered while trying to start extrusion. Find Calvin. "
      |     while 1==1:
      |       popup(popuptext, title="Extrusion Error Code",blocking=True)
      |       popup(resp1, blocking=True)
      |     end
      |   end
      | end
      | 
      | # this function sends a signal and receives a response
      | # signal is a list of 3 strings, 1 character each. first is u. second is the next character. third is final character
      | def send_serial_signal(signal):
      |   signal2char = signal[1]
      |   signal3char = signal[2]
      |   listsignal = [252, get_corr_number(signal2char), get_corr_number(signal3char)]
      |   resp1 = WTSerialBridge.send_command("/dev/ttyUSB0",1200, 8, "None", "One", "None", 1000, "None", "None", listsignal, True)
      |   return resp1
      | end
      | 
      | # this function converts a letter into its ascii number
      | def get_corr_number(letter):
      |   if letter == "A":
